// TwinCAT 3 PLC project TS_PLC
// ProgramVersion: 3.1.4024.0
// libraries:
//   Tc2_Standard, * (Beckhoff Automation GmbH)
//   Tc2_System, * (Beckhoff Automation GmbH)
//   Tc3_Module, * (Beckhoff Automation GmbH)
// project tree:
//   GVLs/ GVL_IO.TcGVL
//   / PlcTask.TcTTO, SimTask.TcTTO
//   POUs/FBs/ FB_Conveyor.TcPOU, FB_Init.TcPOU, FB_LTU.TcPOU, FB_MotorUnit.TcPOU, FB_Reader.TcPOU, FB_Stopper.TcPOU
//   POUs/FBs/Homing/ FB_HomingLTU.TcPOU, FB_HomingManager.TcPOU
//   POUs/FBs/Interchange/ FB_TransferChain_LowerToUpper.TcPOU, FB_TransferChain_UpperToLower.TcPOU, FB_TransferCorner_LowerToUpper.TcPOU, FB_TransferCorner_UpperToLower.TcPOU, FB_DirectTransferGreen.TcPOU, FB_DirectTransferOrange.TcPOU
//   POUs/FBs/Scheduler/ FB_Scheduler.TcPOU, FB_Scheduler_Queue.TcPOU, FB_Scheduler_Queue_copy.TcPOU, FB_ThroughputMonitor.TcPOU
//   POUs/FCs/ FB_AutoPlace.TcPOU
//   POUs/ MAIN.TcPOU, PRG_SIM.TcPOU
//   POUs/Simulation/ FB_InjectAfterRelease.TcPOU, FB_SimConveyor.TcPOU, FB_SimLTU.TcPOU, FB_SimReader.TcPOU, FB_SimStopper.TcPOU
// real-time tasks:
//   TASK PlcTask: cycle T#10ms, priority 20, ADS port 350
//   TASK SimTask: cycle T#10ms, priority 1, ADS port 351
// variable links:
//   TS_PLC/TS_PLC Instance <-> TS_PLC/TS_PLC Instance
//     PlcTask Inputs/MAIN.Conv12_6.MotorOK <-> SimTask Outputs/PRG_SIM.SimConv12_6.MotorOK
//     PlcTask Inputs/MAIN.Conv3_9.MotorOK <-> SimTask Outputs/PRG_SIM.SimConv3_9.MotorOK
//     PlcTask Inputs/MAIN.Conv6_12.MotorOK <-> SimTask Outputs/PRG_SIM.SimConv6_12.MotorOK
//     PlcTask Inputs/MAIN.Conv9_3.MotorOK <-> SimTask Outputs/PRG_SIM.SimConv9_3.MotorOK
//     PlcTask Inputs/MAIN.Conv12_6.RunningIn <-> SimTask Outputs/PRG_SIM.SimConv12_6.RunningIn
//     PlcTask Inputs/MAIN.Conv3_9.RunningIn <-> SimTask Outputs/PRG_SIM.SimConv3_9.RunningIn
//     PlcTask Inputs/MAIN.Conv6_12.RunningIn <-> SimTask Outputs/PRG_SIM.SimConv6_12.RunningIn
//     PlcTask Inputs/MAIN.Conv9_3.RunningIn <-> SimTask Outputs/PRG_SIM.SimConv9_3.RunningIn
//     PlcTask Inputs/MAIN.LTU_12_3.MotorOK <-> SimTask Outputs/PRG_SIM.SimLTU12_3.MotorOK
//     PlcTask Inputs/MAIN.LTU_3_6.MotorOK <-> SimTask Outputs/PRG_SIM.SimLTU3_6.MotorOK
//     PlcTask Inputs/MAIN.LTU_6_9.MotorOK <-> SimTask Outputs/PRG_SIM.SimLTU6_9.MotorOK
//     PlcTask Inputs/MAIN.LTU_9_12.MotorOK <-> SimTask Outputs/PRG_SIM.SimLTU9_12.MotorOK
//     PlcTask Inputs/MAIN.LTU_12_3.PosBottomIn <-> SimTask Outputs/PRG_SIM.SimLTU12_3.PosBottom
//     PlcTask Inputs/MAIN.LTU_3_6.PosBottomIn <-> SimTask Outputs/PRG_SIM.SimLTU3_6.PosBottom
//     PlcTask Inputs/MAIN.LTU_6_9.PosBottomIn <-> SimTask Outputs/PRG_SIM.SimLTU6_9.PosBottom
//     PlcTask Inputs/MAIN.LTU_9_12.PosBottomIn <-> SimTask Outputs/PRG_SIM.SimLTU9_12.PosBottom
//     PlcTask Inputs/MAIN.LTU_12_3.PosMidIn <-> SimTask Outputs/PRG_SIM.SimLTU12_3.PosMid
//     PlcTask Inputs/MAIN.LTU_3_6.PosMidIn <-> SimTask Outputs/PRG_SIM.SimLTU3_6.PosMid
//     PlcTask Inputs/MAIN.LTU_6_9.PosMidIn <-> SimTask Outputs/PRG_SIM.SimLTU6_9.PosMid
//     PlcTask Inputs/MAIN.LTU_9_12.PosMidIn <-> SimTask Outputs/PRG_SIM.SimLTU9_12.PosMid
//     PlcTask Inputs/MAIN.LTU_12_3.PosTopIn <-> SimTask Outputs/PRG_SIM.SimLTU12_3.PosTop
//     PlcTask Inputs/MAIN.LTU_3_6.PosTopIn <-> SimTask Outputs/PRG_SIM.SimLTU3_6.PosTop
//     PlcTask Inputs/MAIN.LTU_6_9.PosTopIn <-> SimTask Outputs/PRG_SIM.SimLTU6_9.PosTop
//     PlcTask Inputs/MAIN.LTU_9_12.PosTopIn <-> SimTask Outputs/PRG_SIM.SimLTU9_12.PosTop
//     PlcTask Inputs/MAIN.LTU_12_3.RunningIn <-> SimTask Outputs/PRG_SIM.SimLTU12_3.PushRunning
//     PlcTask Inputs/MAIN.LTU_3_6.RunningIn <-> SimTask Outputs/PRG_SIM.SimLTU3_6.PushRunning
//     PlcTask Inputs/MAIN.LTU_6_9.RunningIn <-> SimTask Outputs/PRG_SIM.SimLTU6_9.PushRunning
//     PlcTask Inputs/MAIN.LTU_9_12.RunningIn <-> SimTask Outputs/PRG_SIM.SimLTU9_12.PushRunning
//     PlcTask Inputs/MAIN.Reader{3..12 step 3}.I_ReaderValue <-> SimTask Outputs/PRG_SIM.SimReader_{3..12 step 3}.ReaderValue  (4 links)
//     SimTask Inputs/PRG_SIM.SimBlue{3..12 step 3}.CarrierIn <-> PlcTask Outputs/MAIN.Reader{3..12 step 3}.Valid  (4 links)
//     SimTask Inputs/PRG_SIM.SimBlue{3..12 step 3}.CmdDown <-> PlcTask Outputs/MAIN.Blue{3..12 step 3}.StopperDown  (4 links)
//     SimTask Inputs/PRG_SIM.SimConv12_6.MotorRun <-> PlcTask Outputs/MAIN.Conv12_6.MotorRun
//     SimTask Inputs/PRG_SIM.SimConv3_9.MotorRun <-> PlcTask Outputs/MAIN.Conv3_9.MotorRun
//     SimTask Inputs/PRG_SIM.SimConv6_12.MotorRun <-> PlcTask Outputs/MAIN.Conv6_12.MotorRun
//     SimTask Inputs/PRG_SIM.SimConv9_3.MotorRun <-> PlcTask Outputs/MAIN.Conv9_3.MotorRun
//     SimTask Inputs/PRG_SIM.SimLTU12_3.CmdPush <-> PlcTask Outputs/MAIN.LTU_12_3.LTU_MotorRun
//     SimTask Inputs/PRG_SIM.SimLTU3_6.CmdPush <-> PlcTask Outputs/MAIN.LTU_3_6.LTU_MotorRun
//     SimTask Inputs/PRG_SIM.SimLTU6_9.CmdPush <-> PlcTask Outputs/MAIN.LTU_6_9.LTU_MotorRun
//     SimTask Inputs/PRG_SIM.SimLTU9_12.CmdPush <-> PlcTask Outputs/MAIN.LTU_9_12.LTU_MotorRun
//     SimTask Inputs/PRG_SIM.SimLTU12_3.MoveDown <-> PlcTask Outputs/MAIN.LTU_12_3.CylToBottom
//     SimTask Inputs/PRG_SIM.SimLTU3_6.MoveDown <-> PlcTask Outputs/MAIN.LTU_3_6.CylToBottom
//     SimTask Inputs/PRG_SIM.SimLTU6_9.MoveDown <-> PlcTask Outputs/MAIN.LTU_6_9.CylToBottom
//     SimTask Inputs/PRG_SIM.SimLTU9_12.MoveDown <-> PlcTask Outputs/MAIN.LTU_9_12.CylToBottom
//     SimTask Inputs/PRG_SIM.SimLTU12_3.MoveUp <-> PlcTask Outputs/MAIN.LTU_12_3.CylToTop
//     SimTask Inputs/PRG_SIM.SimLTU3_6.MoveUp <-> PlcTask Outputs/MAIN.LTU_3_6.CylToTop
//     SimTask Inputs/PRG_SIM.SimLTU6_9.MoveUp <-> PlcTask Outputs/MAIN.LTU_6_9.CylToTop
//     SimTask Inputs/PRG_SIM.SimLTU9_12.MoveUp <-> PlcTask Outputs/MAIN.LTU_9_12.CylToTop
//     SimTask Inputs/PRG_SIM.SimPurp3_9_1.CmdDown <-> PlcTask Outputs/MAIN.Purple3_9_1.StopperDown
//     SimTask Inputs/PRG_SIM.SimPurp3_9_2.CmdDown <-> PlcTask Outputs/MAIN.Purple3_9_2.StopperDown
//     SimTask Inputs/PRG_SIM.SimPurp9_3_1.CmdDown <-> PlcTask Outputs/MAIN.Purple9_3_1.StopperDown
//     SimTask Inputs/PRG_SIM.SimPurp9_3_2.CmdDown <-> PlcTask Outputs/MAIN.Purple9_3_2.StopperDown
//     SimTask Inputs/PRG_SIM.SimReader_{3..12 step 3}.TriggerRead <-> PlcTask Outputs/MAIN.Reader{3..12 step 3}.vTrigger  (4 links)

CONFIGURATION TS_PLC
    RESOURCE PLC ON TwinCAT3
        TASK PlcTask(INTERVAL := T#10ms, PRIORITY := 20);
        TASK SimTask(INTERVAL := T#10ms, PRIORITY := 1);
        PROGRAM MAIN WITH PlcTask : MAIN;
        PROGRAM PRG_SIM WITH SimTask : PRG_SIM;
    END_RESOURCE
END_CONFIGURATION

// ---- GVLs/GVL_IO.TcGVL
{attribute 'qualified_only'}
VAR_GLOBAL
	//
END_VAR

// ---- POUs/MAIN.TcPOU
PROGRAM MAIN
VAR
	InitFB : FB_Init;
	
	Conv12_6 : FB_Conveyor;
	Conv6_12 : FB_Conveyor;
	Conv3_9 : FB_Conveyor;
	Conv9_3 : FB_Conveyor;
	
	Blue12 : FB_Stopper;
	Blue6 : FB_Stopper;
	Blue3 : FB_Stopper;
	Blue9 : FB_Stopper;
	
	LTU_12_3 : FB_LTU;
	LTU_3_6 : FB_LTU;
	LTU_6_9 : FB_LTU;
	LTU_9_12 : FB_LTU;
	
	Purple9_3_1 : FB_Stopper;
	Purple9_3_2 : FB_Stopper;
	Purple3_9_1 : FB_Stopper;
	Purple3_9_2 : FB_Stopper;
	
	Reader12 : FB_Reader;
	Reader3 : FB_Reader;
	Reader6 : FB_Reader;
	Reader9 : FB_Reader;
	tPulse : TP;
	tPulse1 : TP;
	startRead: BOOL;
	
	
	Blue12_Occupied: BOOL;
	LTU_3_6_LightBarrierIn: BOOL;
	LTU_12_3_LightBarrierIn: BOOL;
	
	Blue6_Occupied: BOOL;
	LTU_6_9_LightBarrierIn: BOOL;
	LTU_9_12_LightBarrierIn: BOOL;
	
	
	Blue9_Occupied: BOOL;
	Purple9_3_1_Occ: BOOL;
	Purple9_3_2_Occ: BOOL;
	
	//Scheduler : FB_Scheduler;
	Scheduler : FB_Scheduler_Queue;
	
	Transfer_12_6 : FB_DirectTransferGreen;
	Transfer_6_12 : FB_DirectTransferGreen;
	
	Transfer_9_3 : FB_DirectTransferOrange;
	Transfer_3_9 : FB_DirectTransferOrange;
	
	Transfer_12_3 : FB_TransferCorner_LowerToUpper;
	Transfer_6_9 : FB_TransferCorner_LowerToUpper;
	Transfer_3_6 : FB_TransferCorner_UpperToLower;
	Transfer_9_12 : FB_TransferCorner_UpperToLower;
	
	Transfer_12_9 : FB_TransferChain_LowerToUpper;
	Transfer_6_3 : FB_TransferChain_LowerToUpper;
	Transfer_9_6 : FB_TransferChain_UpperToLower;
	Transfer_3_12 : FB_TransferChain_UpperToLower;
	
	Throughput : FB_ThroughputMonitor;
	HomingMgr : FB_HomingManager;
	
	DebugWhoWroteBlue6: STRING(128);
	AllLTUsHomed: BOOL;
	HomingError: BOOL;
	ResetGlobal: BOOL;
	SchedulerBusy: BOOL;
	SchedulerQCount: INT;
	StartHomingGlobal: BOOL;
	OnTimer : ton;
	Start: BOOL;
	Auto_Reader12 : FB_AutoPlace;
END_VAR

InitFB(
    Reset     := ,   // manual reset button/flag
    Blue12    := Blue12,
    Blue3     := Blue3,
    Blue6     := Blue6,
    Blue9     := Blue9,
    Purple9_3_1 := Purple9_3_1,
    Purple9_3_2 := Purple9_3_2,
    Purple3_9_1 := Purple3_9_1,
    Purple3_9_2 := Purple3_9_2,
    LTU_12_3 := LTU_12_3,
    LTU_3_6  := LTU_3_6,
    LTU_6_9  := LTU_6_9,
    LTU_9_12 := LTU_9_12,
    Scheduler := Scheduler
);
IF AllLTUsHomed THEN
	Auto_Reader12(BlueStopper:= Blue12.CmdDown, Reader_Trigger=> Reader12.TriggerRead);
END_IF
Conv12_6(
	CmdRunRequest:= TRUE, 
	MotorOK:= , 
	RunningIn:= , 
	PathClear:= TRUE, 
	MotorRun=> , 
	IsRunning=> );
	
Conv6_12(
	CmdRunRequest:= TRUE, 
	MotorOK:= , 
	RunningIn:= , 
	PathClear:= TRUE, 
	MotorRun=> , 
	IsRunning=> );

Conv3_9(
	CmdRunRequest:= TRUE, 
	MotorOK:= , 
	RunningIn:= , 
	PathClear:= TRUE, 
	MotorRun=> , 
	IsRunning=> );
	
Conv9_3(
	CmdRunRequest:= TRUE, 
	MotorOK:= , 
	RunningIn:= , 
	PathClear:= TRUE, 
	MotorRun=> , 
	IsRunning=> );


	
Blue12(CmdDown:= , OccupiedIn:= , StopperDown=> , Occupied=> );
Blue6(CmdDown:= , OccupiedIn:= , StopperDown=> , Occupied=> );
Blue3(CmdDown:= , OccupiedIn:= , StopperDown=> , Occupied=> );
Blue9(CmdDown:= , OccupiedIn:= , StopperDown=> , Occupied=> );

LTU_12_3(
	CmdMoveUp:= , 
	CmdMoveDown:= ,  
	MotorOK:= , 
	RunningIn:= , 
	LightBarrierIn:= , 
	PosBottomIn:= , 
	PosMidIn:= , 
	PosTopIn:= , 
	CylToTop=> , 
	CylToBottom=> , 
	LTU_MotorRun=> , 
	IsRunning=> , 
	PosBottom=> , 
	PosMid=> , 
	PosTop=> , 
	IsFree=> );
	
LTU_3_6(
	CmdMoveUp:= , 
	CmdMoveDown:= ,  
	MotorOK:= , 
	RunningIn:= , 
	LightBarrierIn:= , 
	PosBottomIn:= , 
	PosMidIn:= , 
	PosTopIn:= , 
	CylToTop=> , 
	CylToBottom=> , 
	LTU_MotorRun=> , 
	IsRunning=> , 
	PosBottom=> , 
	PosMid=> , 
	PosTop=> , 
	IsFree=> );
LTU_6_9(
	CmdMoveUp:= , 
	CmdMoveDown:= ,  
	MotorOK:= , 
	RunningIn:= , 
	LightBarrierIn:= , 
	PosBottomIn:= , 
	PosMidIn:= , 
	PosTopIn:= , 
	CylToTop=> , 
	CylToBottom=> , 
	LTU_MotorRun=> , 
	IsRunning=> , 
	PosBottom=> , 
	PosMid=> , 
	PosTop=> , 
	IsFree=> );
LTU_9_12(
	CmdMoveUp:= , 
	CmdMoveDown:= ,  
	MotorOK:= , 
	RunningIn:= , 
	LightBarrierIn:= , 
	PosBottomIn:= , 
	PosMidIn:= , 
	PosTopIn:= , 
	CylToTop=> , 
	CylToBottom=> , 
	LTU_MotorRun=> , 
	IsRunning=> , 
	PosBottom=> , 
	PosMid=> , 
	PosTop=> , 
	IsFree=> );
	
Purple9_3_1(CmdDown:= , OccupiedIn:= , StopperDown=> , Occupied=> );
Purple9_3_2(CmdDown:= , OccupiedIn:= , StopperDown=> , Occupied=> );
Purple3_9_1(CmdDown:= , OccupiedIn:= , StopperDown=> , Occupied=> );
Purple3_9_2(CmdDown:= , OccupiedIn:= , StopperDown=> , Occupied=> );	

	
Reader12(TriggerRead:= ,Dest:=6,Source:=12, ReaderValue=> , Valid=> );	
Reader3(TriggerRead:= ,Dest:=6,Source:=3, ReaderValue=> , Valid=> );	
Reader6(TriggerRead:= ,Dest:=9,Source:=6, ReaderValue=> , Valid=> );	
Reader9(TriggerRead:= ,Dest:=6,Source:=9, ReaderValue=> , Valid=> );	

// === Homing Manager ===
HomingMgr(
    StartHoming := StartHomingGlobal,   // your button / auto-start flag
    Reset       := ,         // global reset button

    LTU_12_3_PosTop    := LTU_12_3.PosTop,
    LTU_12_3_PosBottom := LTU_12_3.PosBottom,
    LTU_12_3_PosMid    := LTU_12_3.PosMid,
    LTU_12_3_Running   := LTU_12_3.IsRunning,

    LTU_3_6_PosTop    := LTU_3_6.PosTop,
    LTU_3_6_PosBottom := LTU_3_6.PosBottom,
    LTU_3_6_PosMid    := LTU_3_6.PosMid,
    LTU_3_6_Running   := LTU_3_6.IsRunning,

    LTU_9_12_PosTop    := LTU_9_12.PosTop,
    LTU_9_12_PosBottom := LTU_9_12.PosBottom,
    LTU_9_12_PosMid    := LTU_9_12.PosMid,
    LTU_9_12_Running   := LTU_9_12.IsRunning,

    LTU_6_9_PosTop    := LTU_6_9.PosTop,
    LTU_6_9_PosBottom := LTU_6_9.PosBottom,
    LTU_6_9_PosMid    := LTU_6_9.PosMid,
    LTU_6_9_Running   := LTU_6_9.IsRunning,

    LTU_12_3_CmdMoveUp   => LTU_12_3.CmdMoveUp,
    LTU_12_3_CmdMoveDown => LTU_12_3.CmdMoveDown,

    LTU_3_6_CmdMoveUp   => LTU_3_6.CmdMoveUp,
    LTU_3_6_CmdMoveDown => LTU_3_6.CmdMoveDown,

    LTU_9_12_CmdMoveUp   => LTU_9_12.CmdMoveUp,
    LTU_9_12_CmdMoveDown => LTU_9_12.CmdMoveDown,

    LTU_6_9_CmdMoveUp   => LTU_6_9.CmdMoveUp,
    LTU_6_9_CmdMoveDown => LTU_6_9.CmdMoveDown,

    AllDone   => AllLTUsHomed,
    AnyError  => HomingError
);

// === Scheduler (enabled only after homing) ===
IF AllLTUsHomed AND NOT HomingError THEN
    Scheduler(
        Reader12_Valid := Reader12.Valid,
        Reader12_Value := Reader12.ReaderValue,
        Reader3_Valid  := Reader3.Valid,
        Reader3_Value  := Reader3.ReaderValue,
        Reader6_Valid  := Reader6.Valid,
        Reader6_Value  := Reader6.ReaderValue,
        Reader9_Valid  := Reader9.Valid,
        Reader9_Value  := Reader9.ReaderValue,

        // Done flags from all transfers
        T12_6_Done := Transfer_12_6.Done,
        T6_12_Done := Transfer_6_12.Done,
        T9_3_Done  := Transfer_9_3.Done,
        T3_9_Done  := Transfer_3_9.Done,
        T12_3_Done := Transfer_12_3.Done,
        T6_9_Done  := Transfer_6_9.Done,
        T3_6_Done  := Transfer_3_6.Done,
        T9_12_Done := Transfer_9_12.Done,
        T12_9_Done := Transfer_12_9.Done,
        T6_3_Done  := Transfer_6_3.Done,
        T9_6_Done  := Transfer_9_6.Done,
        T3_12_Done := Transfer_3_12.Done,

        Reset := 
    );
ELSE
    // Prevent scheduler outputs until homed
    SchedulerBusy := FALSE;
END_IF


// Scheduler -- Only start a transfer if the system is free (no other active transfer)
// Run Scheduler
//Scheduler(
//    Reader12_Valid := Reader12.Valid,
//    Reader12_Value := Reader12.ReaderValue,
//    Reader3_Valid  := Reader3.Valid,
//    Reader3_Value  := Reader3.ReaderValue,
//    Reader6_Valid  := Reader6.Valid,
//    Reader6_Value  := Reader6.ReaderValue,
//    Reader9_Valid  := Reader9.Valid,
//    Reader9_Value  := Reader9.ReaderValue,

//    // pass Done flags from all transfer FBs
//    T12_6_Done := Transfer_12_6.Done,
//    T6_12_Done := Transfer_6_12.Done,
//    T9_3_Done  := Transfer_9_3.Done,
//    T3_9_Done  := Transfer_3_9.Done,
//    T12_3_Done := Transfer_12_3.Done,
//    T6_9_Done  := Transfer_6_9.Done,
//    T3_6_Done  := Transfer_3_6.Done,
//    T9_12_Done := Transfer_9_12.Done,
//    T12_9_Done := Transfer_12_9.Done,
//    T6_3_Done  := Transfer_6_3.Done,
//    T9_6_Done  := Transfer_9_6.Done,
//    T3_12_Done := Transfer_3_12.Done,

//    Reset := 
//);



CASE Scheduler.activeRoute OF
	//..................*** Direct Transfer Green or Lower
	126:Transfer_12_6(JobID := Scheduler.JobID_12_6,
		StartRequest := Scheduler.Start_12_6,
		LTU1_PosOK   := LTU_12_3.PosBottom,
		LTU1_Running := LTU_12_3.IsRunning,
		LTU1_LB      := LTU_12_3_LightBarrierIn,
		LTU2_PosOK   := LTU_3_6.PosBottom,
		LTU2_Running := LTU_3_6.IsRunning,
		LTU2_LB      := LTU_3_6_LightBarrierIn,
		BlueOcc      := Blue12_Occupied,
	
		BlueCmdDown  => Blue12.CmdDown,
		Done         => ,
		Error        => ,
		LTU1_MoveDown=> LTU_12_3.CmdMoveDown,
		LTU2_MoveDown=>	LTU_3_6.CmdMoveDown,
	);
	612:Transfer_6_12(JobID := Scheduler.JobID_6_12,
		StartRequest := Scheduler.Start_6_12,
		LTU1_PosOK   := LTU_6_9.PosBottom,
		LTU1_Running := LTU_6_9.IsRunning,
		LTU1_LB      := LTU_6_9_LightBarrierIn,
		LTU2_PosOK   := LTU_9_12.PosBottom,
		LTU2_Running := LTU_9_12.IsRunning,
		LTU2_LB      := LTU_9_12_LightBarrierIn,
		BlueOcc      := Blue6_Occupied,
	
		BlueCmdDown  => Blue6.CmdDown,
		Done         => ,
		Error        => ,
		LTU1_MoveDown=> LTU_6_9.CmdMoveDown,
		LTU2_MoveDown=>	LTU_9_12.CmdMoveDown
	);
	DebugWhoWroteBlue6 := 'Transfer_6_12';
	//.................*** Direct Transfer Orange or Upper
	93:Transfer_9_3(JobID := Scheduler.JobID_9_3,
		StartRequest:= Scheduler.Start_9_3, 
		LTU1_PosOK:= LTU_9_12.PosTop, 
		LTU1_Running:= LTU_9_12.IsRunning, 
		LTU1_LB:= LTU_9_12_LightBarrierIn, 
		LTU2_PosOK:= LTU_12_3.PosTop, 
		LTU2_Running:= LTU_12_3.IsRunning, 
		LTU2_LB:= LTU_12_3_LightBarrierIn, 
		BlueOcc:= Blue9_Occupied, 
		Purple1Occ:= Purple9_3_1_Occ, 
		Purple2Occ:= Purple9_3_2_Occ, 
		reset:= , 
		BlueCmdDown=> Blue9.CmdDown, 
		Purple1CmdDown=> Purple9_3_1.CmdDown, 
		Purple2CmdDown=> Purple9_3_2.CmdDown, 
		LTU1_MoveUp=> LTU_9_12.CmdMoveUp, 
		LTU2_MoveUp=> LTU_12_3.CmdMoveUp, 
		Done=> , 
		Error=> 
	);
	
	39:Transfer_3_9(JobID := Scheduler.JobID_3_9,
		StartRequest := Scheduler.Start_3_9,
	
		// LTU_3_6
		LTU1_PosOK   := LTU_3_6.PosTop,
		LTU1_Running := LTU_3_6.IsRunning,
		LTU1_LB      := LTU_3_6.LightBarrierIn,
	
		// LTU_6_9
		LTU2_PosOK   := LTU_6_9.PosTop,
		LTU2_Running := LTU_6_9.IsRunning,
		LTU2_LB      := LTU_6_9.LightBarrierIn,
	
		// Stoppers
		BlueOcc      := Blue3.OccupiedIn,
		Purple1Occ   := Purple3_9_1.OccupiedIn,
		Purple2Occ   := Purple3_9_2.OccupiedIn,
	
		reset        := ,
	
		// Outputs
		BlueCmdDown   => Blue3.CmdDown,
		Purple1CmdDown=> Purple3_9_1.CmdDown,
		Purple2CmdDown=> Purple3_9_2.CmdDown,
		LTU1_MoveUp   => LTU_3_6.CmdMoveUp,
		LTU2_MoveUp   => LTU_6_9.CmdMoveUp,
	
		Done  => ,
		Error => 
	);
	
	//.........*************lower to upper corner****************
	123:Transfer_12_3(JobID := Scheduler.JobID_12_3,
		StartRequest:= Scheduler.Start_12_3, 
		LTU_PosTop:= LTU_12_3.PosTop, 
		LTU_PosBottom:= LTU_12_3.PosBottom, 
		LTU_Running:= LTU_12_3.IsRunning, 
		LTU_LB:= LTU_12_3.LightBarrierIn, 
		BlueOcc:= Blue12.OccupiedIn, 
		PurpleOcc:= Purple9_3_2.OccupiedIn, 
		reset:= , 
		BlueCmdDown=> Blue12.CmdDown, 
		PurpleCmdDown=> Purple9_3_2.CmdDown, 
		LTU_MoveUp=> LTU_12_3.CmdMoveUp, 
		LTU_MoveDown=> LTU_12_3.CmdMoveDown, 
		LTU_CmdPush=> LTU_12_3.CmdRun, 
		Done=> , 
		Error=> );
		
	69:Transfer_6_9(JobID := Scheduler.JobID_6_9,
		StartRequest := Scheduler.Start_6_9,
	
		// LTU_6_9
		LTU_PosTop    := LTU_6_9.PosTop,
		LTU_PosBottom := LTU_6_9.PosBottom,
		LTU_Running   := LTU_6_9.IsRunning,
		LTU_LB        := LTU_6_9.LightBarrierIn,
	
		// Stoppers
		BlueOcc       := Blue6.OccupiedIn,
		PurpleOcc     := Purple3_9_2.OccupiedIn,
	
		reset         := ,
	
		// Outputs
		BlueCmdDown   => Blue6.CmdDown,
		PurpleCmdDown => Purple3_9_2.CmdDown,
		LTU_MoveUp    => LTU_6_9.CmdMoveUp,
		LTU_MoveDown  => LTU_6_9.CmdMoveDown,
		LTU_CmdPush   => LTU_6_9.CmdRun,
	
		Done          => ,
		Error         => 
	);
	DebugWhoWroteBlue6 := 'Transfer_6_9';
	//...........**************Upper to Lower Corner.............................
	36:Transfer_3_6(JobID := Scheduler.JobID_3_6,
		StartRequest  := Scheduler.Start_3_6,
	
		LTU_PosTop    := LTU_3_6.PosTop,
		LTU_PosBottom := LTU_3_6.PosBottom,
		LTU_Running   := LTU_3_6.IsRunning,
		LTU_LB        := LTU_3_6.LightBarrierIn,
	
		BlueOcc       := Blue3.OccupiedIn,
		PurpleOcc     := Purple3_9_1.OccupiedIn,
	
		reset         := ,             // or leave blank if you handle reset elsewhere
	
		BlueCmdDown   => Blue3.CmdDown,
		PurpleCmdDown => Purple3_9_1.CmdDown,
		LTU_MoveUp    => LTU_3_6.CmdMoveUp,
		LTU_MoveDown  => LTU_3_6.CmdMoveDown,
		LTU_CmdPush   => LTU_3_6.CmdRun,
	
		Done          => ,
		Error         => 
	);
	912:Transfer_9_12(JobID := Scheduler.JobID_9_12,
		StartRequest  := Scheduler.Start_9_12,
	
		LTU_PosTop    := LTU_9_12.PosTop,
		LTU_PosBottom := LTU_9_12.PosBottom,
		LTU_Running   := LTU_9_12.IsRunning,
		LTU_LB        := LTU_9_12.LightBarrierIn,
	
		BlueOcc       := Blue9.OccupiedIn,
		PurpleOcc     := Purple9_3_1.OccupiedIn,
	
		reset         := ,   // or hook up your reset signal
	
		BlueCmdDown   => Blue9.CmdDown,
		PurpleCmdDown => Purple9_3_1.CmdDown,
		LTU_MoveUp    => LTU_9_12.CmdMoveUp,
		LTU_MoveDown  => LTU_9_12.CmdMoveDown,
		LTU_CmdPush   => LTU_9_12.CmdRun,
	
		Done          => ,
		Error         => 
	);
	
	
	// ............ Multi-hop transfer (12 -> 9) .............................
	//.......Lower to Upper Chain transfer....................................
	129:Transfer_12_9(JobID := Scheduler.JobID_12_9,
		StartRequest  := Scheduler.Start_12_9,
		reset         := ,
	
		// Blue12
		BlueOcc       := Blue12.OccupiedIn,
	
		// LTU_12_3
		LTU1_PosBottom:= LTU_12_3.PosBottom,
		LTU1_PosTop   := LTU_12_3.PosTop,
		LTU1_Running  := LTU_12_3.IsRunning,
		LTU1_LB       := LTU_12_3.LightBarrierIn,
	
		// LTU_3_6
		LTU2_PosBottom:= LTU_3_6.PosBottom,
		LTU2_PosTop   := LTU_3_6.PosTop,
		LTU2_Running  := LTU_3_6.IsRunning,
		LTU2_LB       := LTU_3_6.LightBarrierIn,
	
		// LTU_6_9
		LTU3_PosBottom:= LTU_6_9.PosBottom,
		LTU3_PosTop   := LTU_6_9.PosTop,
		LTU3_Running  := LTU_6_9.IsRunning,
		LTU3_LB       := LTU_6_9.LightBarrierIn,
	
		// Purples
		Purple1_Occ   := Purple9_3_2.OccupiedIn,   // first purple in chain
		Purple2_Occ   := Purple3_9_1.OccupiedIn,   // middle purple
		Purple3_Occ   := Purple3_9_2.OccupiedIn,   // final purple at exit
	
		// Outputs
		BlueCmdDown   => Blue12.CmdDown,
		Purple1CmdDown=> Purple9_3_2.CmdDown,
		Purple2CmdDown=> Purple3_9_1.CmdDown,
		Purple3CmdDown=> Purple3_9_2.CmdDown,
	
		LTU1_CmdPush  => LTU_12_3.CmdRun,
		LTU1_MoveUp   => LTU_12_3.CmdMoveUp,
		LTU1_MoveDown => LTU_12_3.CmdMoveDown,
	
		LTU2_CmdPush  => LTU_3_6.CmdRun,
		LTU2_MoveUp   => LTU_3_6.CmdMoveUp,
		LTU2_MoveDown => LTU_3_6.CmdMoveDown,
	
		LTU3_CmdPush  => LTU_6_9.CmdRun,
		LTU3_MoveUp   => LTU_6_9.CmdMoveUp,
		LTU3_MoveDown => LTU_6_9.CmdMoveDown,
	
		Done          => ,
		Error         => 
	);
	63:Transfer_6_3(JobID := Scheduler.JobID_6_3,
		StartRequest  := Scheduler.Start_6_3,
		reset         := ,
	
		// Blue6
		BlueOcc       := Blue6.OccupiedIn,
	
		// LTU_6_9
		LTU1_PosBottom:= LTU_6_9.PosBottom,
		LTU1_PosTop   := LTU_6_9.PosTop,
		LTU1_Running  := LTU_6_9.IsRunning,
		LTU1_LB       := LTU_6_9.LightBarrierIn,
	
		// LTU_9_12
		LTU2_PosBottom:= LTU_9_12.PosBottom,
		LTU2_PosTop   := LTU_9_12.PosTop,
		LTU2_Running  := LTU_9_12.IsRunning,
		LTU2_LB       := LTU_9_12.LightBarrierIn,
	
		// LTU_12_3
		LTU3_PosBottom:= LTU_12_3.PosBottom,
		LTU3_PosTop   := LTU_12_3.PosTop,
		LTU3_Running  := LTU_12_3.IsRunning,
		LTU3_LB       := LTU_12_3.LightBarrierIn,
	
		// Purples
		Purple1_Occ   := Purple3_9_2.OccupiedIn,
		Purple2_Occ   := Purple9_3_1.OccupiedIn,
		Purple3_Occ   := Purple9_3_2.OccupiedIn,
	
		// Outputs
		BlueCmdDown   => Blue6.CmdDown,
		Purple1CmdDown=> Purple3_9_2.CmdDown,
		Purple2CmdDown=> Purple9_3_1.CmdDown,
		Purple3CmdDown=> Purple9_3_2.CmdDown,
	
		LTU1_CmdPush  => LTU_6_9.CmdRun,
		LTU1_MoveUp   => LTU_6_9.CmdMoveUp,
		LTU1_MoveDown => LTU_6_9.CmdMoveDown,
	
		LTU2_CmdPush  => LTU_9_12.CmdRun,
		LTU2_MoveUp   => LTU_9_12.CmdMoveUp,
		LTU2_MoveDown => LTU_9_12.CmdMoveDown,
	
		LTU3_CmdPush  => LTU_12_3.CmdRun,
		LTU3_MoveUp   => LTU_12_3.CmdMoveUp,
		LTU3_MoveDown => LTU_12_3.CmdMoveDown,
	
		Done          => ,
		Error         => 
	);
	DebugWhoWroteBlue6 := 'Transfer_6_3';
	
	//.......Upper to Lower Chain transfer....................................
	96:Transfer_9_6(JobID := Scheduler.JobID_9_6,
		StartRequest  := Scheduler.Start_9_6,
		reset         := ,
	
		// Blue9
		BlueOcc       := Blue9.OccupiedIn,
	
		// LTU_9_12
		LTU1_PosBottom:= LTU_9_12.PosBottom,
		LTU1_PosTop   := LTU_9_12.PosTop,
		LTU1_Running  := LTU_9_12.IsRunning,
		LTU1_LB       := LTU_9_12.LightBarrierIn,
	
		// LTU_12_3
		LTU2_PosBottom:= LTU_12_3.PosBottom,
		LTU2_PosTop   := LTU_12_3.PosTop,
		LTU2_Running  := LTU_12_3.IsRunning,
		LTU2_LB       := LTU_12_3.LightBarrierIn,
	
		// LTU_3_6
		LTU3_PosBottom:= LTU_3_6.PosBottom,
		LTU3_PosTop   := LTU_3_6.PosTop,
		LTU3_Running  := LTU_3_6.IsRunning,
		LTU3_LB       := LTU_3_6.LightBarrierIn,
	
		// Purples
		Purple1_Occ   := Purple9_3_1.OccupiedIn,   // first purple in path
		Purple2_Occ   := Purple9_3_2.OccupiedIn,   // second purple
	
		// Outputs
		BlueCmdDown   => Blue9.CmdDown,
		Purple1CmdDown=> Purple9_3_1.CmdDown,
		Purple2CmdDown=> Purple9_3_2.CmdDown,
	
		LTU1_CmdPush  => LTU_9_12.CmdRun,
		LTU1_MoveUp   => LTU_9_12.CmdMoveUp,
		LTU1_MoveDown => LTU_9_12.CmdMoveDown,
	
		LTU2_CmdPush  => LTU_12_3.CmdRun,
		LTU2_MoveUp   => LTU_12_3.CmdMoveUp,
		LTU2_MoveDown => LTU_12_3.CmdMoveDown,
	
		LTU3_CmdPush  => LTU_3_6.CmdRun,
		LTU3_MoveUp   => LTU_3_6.CmdMoveUp,
		LTU3_MoveDown => LTU_3_6.CmdMoveDown,
	
		Done          => ,
		Error         => 
	);	
	312:Transfer_3_12(JobID := Scheduler.JobID_3_12,
		StartRequest  := Scheduler.Start_3_12,
		reset         := ,
	
		// Blue3
		BlueOcc       := Blue3.OccupiedIn,
	
		// LTU_3_6
		LTU1_PosBottom:= LTU_3_6.PosBottom,
		LTU1_PosTop   := LTU_3_6.PosTop,
		LTU1_Running  := LTU_3_6.IsRunning,
		LTU1_LB       := LTU_3_6.LightBarrierIn,
	
		// LTU_6_9
		LTU2_PosBottom:= LTU_6_9.PosBottom,
		LTU2_PosTop   := LTU_6_9.PosTop,
		LTU2_Running  := LTU_6_9.IsRunning,
		LTU2_LB       := LTU_6_9.LightBarrierIn,
	
		// LTU_9_12
		LTU3_PosBottom:= LTU_9_12.PosBottom,
		LTU3_PosTop   := LTU_9_12.PosTop,
		LTU3_Running  := LTU_9_12.IsRunning,
		LTU3_LB       := LTU_9_12.LightBarrierIn,
	
		// Purples
		Purple1_Occ   := Purple3_9_1.OccupiedIn,
		Purple2_Occ   := Purple3_9_2.OccupiedIn,
		Purple3_Occ   := Purple9_3_1.OccupiedIn,
	
		// Outputs
		BlueCmdDown   => Blue3.CmdDown,
		Purple1CmdDown=> Purple3_9_1.CmdDown,
		Purple2CmdDown=> Purple3_9_2.CmdDown,
		Purple3CmdDown=> Purple9_3_1.CmdDown,
	
		LTU1_CmdPush  => LTU_3_6.CmdRun,
		LTU1_MoveUp   => LTU_3_6.CmdMoveUp,
		LTU1_MoveDown => LTU_3_6.CmdMoveDown,
	
		LTU2_CmdPush  => LTU_6_9.CmdRun,
		LTU2_MoveUp   => LTU_6_9.CmdMoveUp,
		LTU2_MoveDown => LTU_6_9.CmdMoveDown,
	
		LTU3_CmdPush  => LTU_9_12.CmdRun,
		LTU3_MoveUp   => LTU_9_12.CmdMoveUp,
		LTU3_MoveDown => LTU_9_12.CmdMoveDown,
	
		Done          => ,
		Error         => 
	);
ELSE
    // no active route → don’t call any transfer FB
	//DebugWhoWroteBlue6 := 'NONE';
END_CASE


Throughput(
    DonePulse := (
        Transfer_12_6.Done OR
        Transfer_6_12.Done OR
        Transfer_9_3.Done  OR
        Transfer_3_9.Done  OR
        Transfer_12_3.Done OR
        Transfer_6_9.Done  OR
        Transfer_3_6.Done  OR
        Transfer_9_12.Done OR
        Transfer_12_9.Done OR
        Transfer_6_3.Done  OR
        Transfer_9_6.Done  OR
        Transfer_3_12.Done
    ),
    Reset := 
);

END_PROGRAM

// ---- POUs/FBs/FB_Init.TcPOU
FUNCTION_BLOCK FB_Init
VAR_INPUT
    Reset : BOOL;   // external reset (button/flag)
END_VAR
VAR_IN_OUT
    Blue12, Blue3, Blue6, Blue9 : FB_Stopper;
    Purple9_3_1, Purple9_3_2, Purple3_9_1, Purple3_9_2 : FB_Stopper;
    LTU_12_3, LTU_3_6, LTU_6_9, LTU_9_12 : FB_LTU;
    Scheduler : FB_Scheduler_Queue;
END_VAR
VAR
    firstScan : BOOL := TRUE;   // internal latch
END_VAR

// --- Safe State Logic ---
IF firstScan OR Reset THEN
    // Blue stoppers (all blocking)
    Blue12.CmdDown := TRUE;
    Blue3.CmdDown  := TRUE;
    Blue6.CmdDown  := TRUE;
    Blue9.CmdDown  := TRUE;

    // Purple stoppers (all blocking)
    Purple9_3_1.CmdDown := TRUE;
    Purple9_3_2.CmdDown := TRUE;
    Purple3_9_1.CmdDown := TRUE;
    Purple3_9_2.CmdDown := TRUE;

    // LTUs (all idle)
    LTU_12_3.CmdMoveUp   := FALSE;
    LTU_12_3.CmdMoveDown := FALSE;
    LTU_12_3.CmdRun      := FALSE;

    LTU_3_6.CmdMoveUp    := FALSE;
    LTU_3_6.CmdMoveDown  := FALSE;
    LTU_3_6.CmdRun       := FALSE;

    LTU_6_9.CmdMoveUp    := FALSE;
    LTU_6_9.CmdMoveDown  := FALSE;
    LTU_6_9.CmdRun       := FALSE;

    LTU_9_12.CmdMoveUp   := FALSE;
    LTU_9_12.CmdMoveDown := FALSE;
    LTU_9_12.CmdRun      := FALSE;

    // Tell Scheduler to reset itself
    Scheduler(Reset := TRUE);

    // clear firstScan latch
    firstScan := FALSE;
ELSE
    // normal scheduler call, Reset=FALSE
    Scheduler(Reset := FALSE);
END_IF

END_FUNCTION_BLOCK

// ---- POUs/FBs/FB_Stopper.TcPOU
FUNCTION_BLOCK FB_Stopper
VAR_INPUT
    CmdDown   : BOOL;   // TRUE = stopper down (block carrier)
    OccupiedIn AT%I*: BOOL;   // Sensor input
END_VAR
VAR_OUTPUT
    StopperDown AT%Q*: BOOL; // Actuator output
    Occupied    : BOOL; // Output copy of sensor
END_VAR

// Direct assignments
StopperDown := CmdDown;
Occupied    := OccupiedIn;

END_FUNCTION_BLOCK

// ---- POUs/FBs/FB_LTU.TcPOU
FUNCTION_BLOCK FB_LTU
VAR_INPUT
    CmdMoveUp      : BOOL;   // request cylinder to Top
    CmdMoveDown    : BOOL;   // request cylinder to Bottom
    CmdRun         : BOOL;   // run LTU motor
    MotorOK        AT%I*: BOOL;
    RunningIn      AT%I*: BOOL;   // motor running feedback
    LightBarrierIn AT%I*: BOOL;   // TRUE if LTU free
    PosBottomIn    AT%I*: BOOL;
    PosMidIn       AT%I*: BOOL;
    PosTopIn       AT%I*: BOOL;
END_VAR
VAR_OUTPUT
    CylToTop       AT%Q*: BOOL;   // actuator output
    CylToBottom    AT%Q*: BOOL;   // actuator output
    LTU_MotorRun   AT%Q*: BOOL;   // actuator output
    IsRunning      : BOOL;   // motor running feedback
    PosBottom      : BOOL;
    PosMid         : BOOL;
    PosTop         : BOOL;
    IsFree         : BOOL;   // derived from LightBarrierIn
END_VAR
VAR
    Motor : FB_MotorUnit;
END_VAR

// Cylinder logic (safe mutual exclusion)
CylToTop    := CmdMoveUp AND NOT CmdMoveDown;
CylToBottom := CmdMoveDown AND NOT CmdMoveUp;

// Motor logic
Motor(CmdRun := CmdRun,
      MotorOK := MotorOK,
      RunningIn := RunningIn);

LTU_MotorRun := Motor.MotorRun;
IsRunning    := Motor.IsRunning;

// Pass-through sensors
PosBottom := PosBottomIn;
PosMid    := PosMidIn;
PosTop    := PosTopIn;
IsFree    := LightBarrierIn;

END_FUNCTION_BLOCK

// ---- POUs/FBs/FB_MotorUnit.TcPOU
FUNCTION_BLOCK FB_MotorUnit
VAR_INPUT
    CmdRun   : BOOL;   // Command from controller
    MotorOK  : BOOL;   // from sensor Motor health input
	RunningIn : BOOL;  // From sensor (conveyor running feedback)
END_VAR
VAR_OUTPUT
    MotorRun : BOOL;   // Output to motor actuator
    IsRunning: BOOL;   // Sensor input: motor running
END_VAR
VAR
    //
END_VAR

// Simple interlock
MotorRun   := CmdRun AND MotorOK ;
IsRunning  := RunningIn;

END_FUNCTION_BLOCK

// ---- POUs/FBs/Scheduler/FB_Scheduler_Queue.TcPOU
FUNCTION_BLOCK FB_Scheduler_Queue
VAR_INPUT
    // Reader inputs
    Reader12_Valid : BOOL;
    Reader12_Value : INT;
    Reader3_Valid  : BOOL;
    Reader3_Value  : INT;
    Reader6_Valid  : BOOL;
    Reader6_Value  : INT;
    Reader9_Valid  : BOOL;
    Reader9_Value  : INT;

    // Done flags from transfers
    T12_6_Done, T6_12_Done : BOOL;
    T9_3_Done,  T3_9_Done  : BOOL;
    T12_3_Done, T6_9_Done  : BOOL;
    T3_6_Done,  T9_12_Done : BOOL;
    T12_9_Done, T6_3_Done  : BOOL;
    T9_6_Done,  T3_12_Done : BOOL;

    Reset : BOOL;
END_VAR
VAR_OUTPUT
    // Start signals (1-scan pulses)
    Start_12_6, Start_6_12 : BOOL;
    Start_9_3,  Start_3_9  : BOOL;
    Start_12_3, Start_6_9  : BOOL;
    Start_3_6,  Start_9_12 : BOOL;
    Start_12_9, Start_6_3  : BOOL;
    Start_9_6,  Start_3_12 : BOOL;

    Busy        : BOOL;
    QCount      : INT;     // number of queued requests
    activeRoute : INT;     // currently executing route
END_VAR
VAR
    queue   : ARRAY[1..10] OF INT;   // FIFO buffer (10 deep)
    head    : INT := 1;
    tail    : INT := 1;
	prevR12, prevR3, prevR6, prevR9 : BOOL;
END_VAR

// === Reset ===
IF Reset THEN
    head := 1; tail := 1; QCount := 0;
    Busy := FALSE; activeRoute := 0;
END_IF

// === Enqueue new reader requests ===
IF Reader12_Valid AND NOT prevR12 THEN
    CASE Reader12_Value OF
        6: Enqueue(126);
        3: Enqueue(123);
        9: Enqueue(129);
    END_CASE
END_IF
prevR12 := Reader12_Valid;

IF Reader6_Valid AND NOT prevR6 THEN
    CASE Reader6_Value OF
        12: Enqueue(612);
        9:  Enqueue(69);
        3:  Enqueue(63);
    END_CASE
END_IF
prevR6 := Reader6_Valid;

IF Reader3_Valid AND NOT prevR3 THEN
    CASE Reader3_Value OF
        9:  Enqueue(39);
        6:  Enqueue(36);
        12: Enqueue(312);
    END_CASE
END_IF
prevR3 := Reader3_Valid;

IF Reader9_Valid AND NOT prevR9 THEN
    CASE Reader9_Value OF
        3:  Enqueue(93);
        12: Enqueue(912);
        6:  Enqueue(96);
    END_CASE
END_IF
prevR9 := Reader9_Valid;


// === Dispatch logic ===
IF NOT Busy AND QCount > 0 THEN
    activeRoute := queue[head];
    head := (head MOD 10) + 1;
    QCount := QCount - 1;
    Busy := TRUE;

    // one-shot Start signal
    CASE activeRoute OF
        126: Start_12_6 := TRUE;
        612: Start_6_12 := TRUE;
        93 : Start_9_3  := TRUE;
        39 : Start_3_9  := TRUE;
        123: Start_12_3 := TRUE;
        69 : Start_6_9  := TRUE;
        36 : Start_3_6  := TRUE;
        912: Start_9_12 := TRUE;
        129: Start_12_9 := TRUE;
        63 : Start_6_3  := TRUE;
        96 : Start_9_6  := TRUE;
        312: Start_3_12 := TRUE;
    END_CASE
ELSE
    Start_12_6 := FALSE; Start_6_12 := FALSE;
    Start_9_3  := FALSE; Start_3_9  := FALSE;
    Start_12_3 := FALSE; Start_6_9  := FALSE;
    Start_3_6  := FALSE; Start_9_12 := FALSE;
    Start_12_9 := FALSE; Start_6_3  := FALSE;
    Start_9_6  := FALSE; Start_3_12 := FALSE;
END_IF


// === Completion check ===
CASE activeRoute OF
    126: IF T12_6_Done THEN Busy := FALSE; activeRoute := 0; END_IF
    612: IF T6_12_Done THEN Busy := FALSE; activeRoute := 0; END_IF
    93 : IF T9_3_Done  THEN Busy := FALSE; activeRoute := 0; END_IF
    39 : IF T3_9_Done  THEN Busy := FALSE; activeRoute := 0; END_IF
    123: IF T12_3_Done THEN Busy := FALSE; activeRoute := 0; END_IF
    69 : IF T6_9_Done  THEN Busy := FALSE; activeRoute := 0; END_IF
    36 : IF T3_6_Done  THEN Busy := FALSE; activeRoute := 0; END_IF
    912: IF T9_12_Done THEN Busy := FALSE; activeRoute := 0; END_IF
    129: IF T12_9_Done THEN Busy := FALSE; activeRoute := 0; END_IF
    63 : IF T6_3_Done  THEN Busy := FALSE; activeRoute := 0; END_IF
    96 : IF T9_6_Done  THEN Busy := FALSE; activeRoute := 0; END_IF
    312: IF T3_12_Done THEN Busy := FALSE; activeRoute := 0; END_IF
END_CASE

METHOD PRIVATE Enqueue : BOOL
VAR_INPUT
    route : INT;
END_VAR

IF QCount < 10 THEN
    queue[tail] := route;
    tail := (tail MOD 10) + 1;
    QCount := QCount + 1;
    Enqueue := TRUE;
ELSE
    Enqueue := FALSE; // queue full
END_IF
END_METHOD

END_FUNCTION_BLOCK

// ---- POUs/FBs/FB_Conveyor.TcPOU
FUNCTION_BLOCK FB_Conveyor
VAR_INPUT
    CmdRunRequest : BOOL;   // scheduler command
    MotorOK       AT%I*: BOOL;   // from sensor
    RunningIn     AT%I*: BOOL;   // from sensor
    PathClear     : BOOL;
END_VAR
VAR_OUTPUT
    MotorRun      AT%Q*: BOOL;   // Output to motor cmd
    IsRunning     : BOOL;
END_VAR
VAR
    Motor : FB_MotorUnit;
END_VAR

Motor(CmdRun := (CmdRunRequest AND PathClear),
      MotorOK := MotorOK,
      RunningIn := RunningIn);

MotorRun  := Motor.MotorRun;
IsRunning := Motor.IsRunning;

END_FUNCTION_BLOCK

// ---- POUs/FBs/FB_Reader.TcPOU
FUNCTION_BLOCK FB_Reader
VAR_INPUT
    TriggerRead : BOOL;   // input from I_ReaderXX_Trigger
	BlueOcc : BOOL;
	ForceDest   : INT := 0; // 0 = random, else fixed destination (12/3/6/9)
	Source : INT;
	Dest : Int;
END_VAR
VAR_OUTPUT
    ReaderValue : INT;    // destination code (12, 3, 6, 9)
    Valid       AT%Q*: BOOL;   // TRUE for one scan when a new value is read
END_VAR
VAR
    lastTrigger : BOOL;
	I_ReaderValue AT%I*:INT;
	vTrigger AT%Q*: BOOL;
    seed        : UDINT := 12345;
    pick        : INT;
END_VAR

// Rising edge detection
IF TriggerRead AND NOT lastTrigger THEN
    IF ForceDest <> 0 THEN
        // Use forced destination
        ReaderValue := ForceDest;
    ELSE
        // Generate random until != Source
        REPEAT
            seed := (1103515245 * seed + 12345);
            CASE (seed MOD 4) OF
                0: pick := 12;
                1: pick := 3;
                2: pick := 6;
                3: pick := 9;
            END_CASE
        UNTIL pick <> Source
        END_REPEAT;
        ReaderValue := pick;
    END_IF
    Valid := TRUE;
ELSE
    Valid := FALSE;
END_IF

lastTrigger := TriggerRead;
//// detect rising edge
//IF TriggerRead AND NOT lastTrigger THEN
//    Valid := TRUE;           // one-cycle pulse
//    ReaderValue := Dest;     // assign destination
//ELSE
//    Valid := FALSE;
//    ReaderValue := 0;
//END_IF

//// update memory
//lastTrigger := TriggerRead;

END_FUNCTION_BLOCK

// ---- POUs/FBs/Interchange/FB_DirectTransferGreen.TcPOU
FUNCTION_BLOCK FB_DirectTransferGreen
VAR_INPUT
    StartRequest : BOOL;   // reader triggered with correct Dest
	JobID        : UDINT;     // unique per dispatch
    LTU1_PosOK   : BOOL;   // e.g. LTU_12_3.PosBottom
    LTU1_Running : BOOL;
    LTU1_LB      : BOOL;   // LightBarrier TRUE=empty
    LTU2_PosOK   : BOOL;   // e.g. LTU_3_6.PosBottom
    LTU2_Running : BOOL;
    LTU2_LB      : BOOL;
    BlueOcc      : BOOL;   // Blue stopper Occupied
END_VAR
VAR_OUTPUT
    BlueCmdDown : BOOL;   // TRUE=block, FALSE=release
	LTU1_MoveDown : BOOL; // True=bottom
	LTU2_MoveDown : BOOL;
	LTU1_MotorRunCmd : BOOL; // True=Run
	LTU2_MotorRunCmd : BOOL;
    Done        : BOOL;
    Error       : BOOL;
END_VAR
VAR
    state    : INT := 0;
    tTimeout : TON;
	reset: BOOL;
	lastRequest: BOOL;
	lastJobID  : UDINT := 0;   // store previous job ID
END_VAR

CASE state OF
0: // IDLE
    BlueCmdDown := TRUE; //Blocking
    Error := FALSE;
	
    // latch Done until new request comes
    IF StartRequest AND JobID <> lastJobID THEN
		// command both LTUs down
        LTU1_MoveDown := TRUE;
        LTU2_MoveDown := TRUE;
        Done := FALSE;        // reset Done on new request
		lastJobID := JobID;
        state := 1;           // start cycle
    END_IF
    

1: // ALIGN
    // keep commanding move down until confirmed
    LTU1_MoveDown := TRUE;
    LTU2_MoveDown := TRUE;

    IF LTU1_PosOK 
       AND LTU2_PosOK  THEN
//        LTU1_MoveDown := FALSE;
//        LTU2_MoveDown := FALSE;
        state := 2; // RELEASE
    END_IF

2: // RELEASE
    IF BlueOcc THEN
        BlueCmdDown := FALSE;   // open for release
        //tTimeout(IN := TRUE, PT := T#8S);
        state := 3;
    END_IF

3: // WAIT_ENTER_LT1
    // Re-block once carrier left Blue
    IF NOT BlueOcc THEN
        BlueCmdDown := TRUE;
    END_IF

    IF NOT LTU1_LB THEN
        state := 4;
//        tTimeout(IN := TRUE, PT := T#8S);
//    ELSIF tTimeout.Q THEN 
//        state := 99; 
    END_IF

4: // WAIT_LEAVE_LT1
	BlueCmdDown := TRUE;//reblock 
	IF LTU1_PosOK 
       AND LTU2_PosOK THEN
		LTU1_MotorRunCmd := TRUE;
		LTU2_MotorRunCmd := TRUE;
	END_IF
    IF LTU1_LB THEN
        state := 5;
//        tTimeout(IN := TRUE, PT := T#8S);
//    ELSIF tTimeout.Q THEN state := 99; 
	END_IF

5: // WAIT_ENTER_LT2
    IF NOT LTU2_LB THEN
        state := 6;
//        tTimeout(IN := TRUE, PT := T#8S);
//    ELSIF tTimeout.Q THEN state := 99; 
	END_IF

6: // WAIT_LEAVE_LT2
    IF LTU2_LB THEN
        BlueCmdDown := TRUE;
        Done := TRUE;
        state := 0;
    //ELSIF tTimeout.Q THEN state := 99; 
	END_IF

99: // ERROR
    BlueCmdDown := TRUE;
    Error := TRUE;
	IF reset THEN
		 state := 0;
	END_IF
   
END_CASE

// --- Edge detection for StartRequest ---
//lastRequest := StartRequest;

END_FUNCTION_BLOCK

// ---- POUs/FBs/Interchange/FB_DirectTransferOrange.TcPOU
FUNCTION_BLOCK FB_DirectTransferOrange
VAR_INPUT
    StartRequest : BOOL;   // reader detected correct dest
	JobID        : UDINT;     // unique per dispatch
    LTU1_PosOK   : BOOL;   // LTU1 at Top
    LTU1_Running : BOOL;
    LTU1_LB      : BOOL;
    LTU2_PosOK   : BOOL;   // LTU2 at Top
    LTU2_Running : BOOL;
    LTU2_LB      : BOOL;
    BlueOcc      : BOOL;   // entry stopper occupied
    Purple1Occ   : BOOL;   // intermediate purple (near LTU1)
    Purple2Occ   : BOOL;   // final purple (exit stopper)
    reset        : BOOL;
END_VAR
VAR_OUTPUT
    BlueCmdDown    : BOOL;
    Purple1CmdDown : BOOL;
    Purple2CmdDown : BOOL;
    LTU1_MoveUp    : BOOL;
    LTU2_MoveUp    : BOOL;
	LTU1_MotorRunCmd : BOOL; // True=bottom
	LTU2_MotorRunCmd : BOOL;
    Done           : BOOL;
    Error          : BOOL;
END_VAR
VAR
    state : INT := 0;
	lastRequest: BOOL;
	lastJobID  : UDINT := 0;   // store previous job ID
END_VAR

CASE state OF
0: // IDLE
    BlueCmdDown    := TRUE;//blocking
    Purple1CmdDown := FALSE;//release
    Purple2CmdDown := FALSE;//release
    Error := FALSE;

    IF StartRequest AND JobID <> lastJobID THEN
        LTU1_MoveUp := TRUE;
        LTU2_MoveUp := TRUE;
		Done := FALSE; 
		lastJobID := JobID;
        state := 1;
    END_IF

1: // ALIGN
    LTU1_MoveUp := TRUE;
    LTU2_MoveUp := TRUE;

    IF LTU1_PosOK AND 
        LTU2_PosOK  THEN
        
        state := 2;
    END_IF

2: // CHECK_PURPLES
    IF (NOT Purple1CmdDown) AND (NOT Purple2CmdDown) THEN
        state := 3;
    END_IF

3: // RELEASE
    IF BlueOcc THEN
        BlueCmdDown := FALSE;
        state := 4;
    END_IF

4: // WAIT_ENTER_LT1
    IF NOT BlueOcc THEN
        BlueCmdDown := TRUE; // re-block entry
    END_IF
	
    IF NOT LTU1_LB THEN
        state := 5;
    END_IF

5: // WAIT_LEAVE_LT1
	BlueCmdDown := TRUE;//reblock 
	LTU1_MotorRunCmd := TRUE;
	LTU2_MotorRunCmd := TRUE;
    IF LTU1_LB THEN
        state := 6;
    END_IF

6: // WAIT_ENTER_LT2
    IF NOT LTU2_LB THEN
        state := 7;
    END_IF

7: // WAIT_LEAVE_LT2
    IF LTU2_LB THEN
        state := 8;
    END_IF

8: // WAIT_AT_PURPLE
    IF Purple2Occ THEN
        Purple2CmdDown := FALSE; // release final carrier
        Done := TRUE;
        state := 0;
    END_IF

99: // ERROR
    BlueCmdDown    := TRUE;
    Purple1CmdDown := TRUE;
    Purple2CmdDown := TRUE;
    Error := TRUE;
    IF reset THEN
        state := 0;
    END_IF
END_CASE

// --- Edge detection for StartRequest ---
lastRequest := StartRequest;

END_FUNCTION_BLOCK

// ---- POUs/FBs/Interchange/FB_TransferCorner_LowerToUpper.TcPOU
FUNCTION_BLOCK FB_TransferCorner_LowerToUpper
VAR_INPUT
    StartRequest : BOOL;   // reader request
	JobID        : UDINT;     // unique per dispatch
    LTU_PosTop   : BOOL;
    LTU_PosBottom: BOOL;
    LTU_Running  : BOOL;   // push motor feedback
    LTU_LB       : BOOL;   // TRUE = empty, FALSE = carrier inside
    BlueOcc      : BOOL;
    PurpleOcc    : BOOL;
    reset        : BOOL;
END_VAR
VAR_OUTPUT
    BlueCmdDown   : BOOL;
    PurpleCmdDown : BOOL;
    LTU_MoveUp    : BOOL;
    LTU_MoveDown  : BOOL;
    LTU_CmdPush   : BOOL;
    Done          : BOOL;
    Error         : BOOL;
END_VAR
VAR
    state : INT := 0;
	lastRequest: BOOL;
	lastJobID  : UDINT := 0;   // store previous job ID
END_VAR

CASE state OF
0: // IDLE
    BlueCmdDown   := TRUE;
    PurpleCmdDown := TRUE;
    LTU_MoveUp    := FALSE;
    LTU_MoveDown  := TRUE;   // stay aligned to Bottom by default
    LTU_CmdPush   := FALSE;
    Error := FALSE;

    // latch Done until a new StartRequest arrives
    IF StartRequest AND JobID <> lastJobID THEN
        Done := FALSE;           // clear done on new request
		lastJobID := JobID;
        state := 1;              // start new transfer
    END_IF

1: // RELEASE BLUE
    IF BlueOcc AND LTU_PosBottom THEN
        BlueCmdDown := FALSE;   // let carrier enter LTU
        state := 2;
    END_IF

2: // WAIT ENTER LTU
    IF NOT BlueOcc THEN
        BlueCmdDown := TRUE;    // re-block entry
    END_IF
    IF NOT LTU_LB THEN          // LTU occupied
        state := 3;
    END_IF

3: // LIFT TO TOP
	BlueCmdDown := TRUE;
    LTU_MoveDown := FALSE;
    LTU_MoveUp   := TRUE;

    IF LTU_PosTop THEN
        LTU_MoveUp := FALSE;
        state := 4;
    END_IF

4: // PUSH OUT
    IF PurpleOcc THEN
        PurpleCmdDown := FALSE;
    END_IF
     
    IF NOT PurpleCmdDown THEN   // only push if exit released
        LTU_CmdPush := TRUE;
        IF PurpleOcc THEN
            LTU_CmdPush := FALSE;
            Done := TRUE;      // latch Done here
            state := 0;        // return to IDLE, but Done stays TRUE
        END_IF
    END_IF

99: // ERROR
    BlueCmdDown   := TRUE;
    PurpleCmdDown := TRUE;
    LTU_MoveUp    := FALSE;
    LTU_MoveDown  := FALSE;
    LTU_CmdPush   := FALSE;
    Error := TRUE;
    IF reset THEN
        state := 0;
    END_IF
END_CASE

// Rising edge detector for StartRequest
lastRequest := StartRequest;

END_FUNCTION_BLOCK

// ---- POUs/FBs/Interchange/FB_TransferCorner_UpperToLower.TcPOU
FUNCTION_BLOCK FB_TransferCorner_UpperToLower
VAR_INPUT
    StartRequest : BOOL;   // request to start
	JobID        : UDINT;     // unique per dispatch
    LTU_PosTop   : BOOL;
    LTU_PosBottom: BOOL;
    LTU_Running  : BOOL;
    LTU_LB       : BOOL;   // TRUE=empty, FALSE=occupied
    BlueOcc      : BOOL;   // Blue entry occupied
    PurpleOcc    : BOOL;   // entry purple occupied (must be released)
    reset        : BOOL;
END_VAR
VAR_OUTPUT
    BlueCmdDown   : BOOL;
    PurpleCmdDown : BOOL;
    LTU_MoveUp    : BOOL;
    LTU_MoveDown  : BOOL;
    LTU_CmdPush   : BOOL;
    Done          : BOOL;
    Error         : BOOL;
END_VAR
VAR
    state : INT := 0;
	lastRequest: BOOL;
	lastJobID  : UDINT := 0;   // store previous job ID
END_VAR

CASE state OF
0: // IDLE
    BlueCmdDown   := TRUE;
    PurpleCmdDown := TRUE;   // block by default
    LTU_MoveUp    := TRUE;   // keep aligned to Top
    LTU_MoveDown  := FALSE;
    LTU_CmdPush   := FALSE;
    Error := FALSE;

    // latch Done until new request comes
    IF StartRequest AND JobID <> lastJobID THEN
        Done := FALSE;        // reset Done on new request
		lastJobID := JobID;
        state := 1;           // start cycle
    END_IF

1: // ALIGN TOP
    LTU_MoveUp := TRUE;
    IF LTU_PosTop AND NOT LTU_Running THEN
        LTU_MoveUp := FALSE;
        state := 2;
    END_IF

2: // RELEASE
    IF BlueOcc AND PurpleCmdDown THEN
        BlueCmdDown := FALSE;  // let carrier into LTU
        state := 3;
    END_IF

3: // WAIT_ENTER_LT
    IF NOT BlueOcc THEN
        BlueCmdDown := TRUE;   // re-block entry
    END_IF
    IF NOT LTU_LB THEN
        state := 4;
    END_IF

4: // LIFT DOWN
	BlueCmdDown := TRUE;//reblock 
    LTU_MoveDown := TRUE;
    IF LTU_PosBottom AND NOT LTU_Running THEN
        LTU_MoveDown := FALSE;
        state := 5;
    END_IF

5: // PUSH OUT
    LTU_CmdPush := TRUE;
    IF LTU_LB THEN  // became empty again
        LTU_CmdPush := FALSE;
        Done := TRUE;         // latch Done
        state := 0;           // go back to IDLE
    END_IF

99: // ERROR
    BlueCmdDown   := TRUE;
    PurpleCmdDown := TRUE;
    LTU_MoveUp    := FALSE;
    LTU_MoveDown  := FALSE;
    LTU_CmdPush   := FALSE;
    Error := TRUE;
    IF reset THEN
        state := 0;
    END_IF
END_CASE

// --- Edge detection for StartRequest ---
lastRequest := StartRequest;

END_FUNCTION_BLOCK

// ---- POUs/FBs/Interchange/FB_TransferChain_LowerToUpper.TcPOU
FUNCTION_BLOCK FB_TransferChain_LowerToUpper
VAR_INPUT
    StartRequest : BOOL;
	JobID        : UDINT;     // unique per dispatch
    reset        : BOOL;

    // Blue12
    BlueOcc      : BOOL;

    // LTU_12_3
    LTU1_PosBottom, LTU1_PosTop, LTU1_Running, LTU1_LB : BOOL;

    // LTU_3_6
    LTU2_PosBottom, LTU2_PosTop, LTU2_Running, LTU2_LB : BOOL;

    // LTU_6_9
    LTU3_PosBottom, LTU3_PosTop, LTU3_Running, LTU3_LB : BOOL;

    // Purple stoppers
    Purple1_Occ : BOOL;   // Purple9_3_2
    Purple2_Occ : BOOL;   // Purple3_9_1
    Purple3_Occ : BOOL;   // Purple3_9_2
END_VAR
VAR_OUTPUT
    // Blue
    BlueCmdDown : BOOL;

    // Purple
    Purple1CmdDown, Purple2CmdDown, Purple3CmdDown : BOOL;

    // LTU_12_3
    LTU1_CmdPush, LTU1_MoveUp, LTU1_MoveDown : BOOL;

    // LTU_3_6
    LTU2_CmdPush, LTU2_MoveUp, LTU2_MoveDown : BOOL;

    // LTU_6_9
    LTU3_CmdPush, LTU3_MoveUp, LTU3_MoveDown : BOOL;

    Done  : BOOL;
    Error : BOOL;
END_VAR
VAR
    state       : INT := 0;
    lastRequest : BOOL := FALSE;
	lastJobID  : UDINT := 0;   // store previous job ID
END_VAR

CASE state OF
0: // IDLE
    BlueCmdDown     := TRUE;
    Purple1CmdDown  := TRUE;
    Purple2CmdDown  := TRUE;
    Purple3CmdDown  := TRUE;
	LTU1_MoveDown := FALSE;
	LTU1_MoveUp := FALSE;
	LTU2_MoveDown := FALSE;
	LTU2_MoveUp := FALSE;
	LTU3_MoveDown := FALSE;
	LTU3_MoveUp := FALSE;
	
	
    LTU1_CmdPush := FALSE;
    LTU2_CmdPush := FALSE;
    LTU3_CmdPush := FALSE;

    Error := FALSE;

    IF StartRequest AND JobID <> lastJobID THEN
        Done := FALSE;
		lastJobID := JobID;
        state := 1;
    END_IF

1: // ALIGN
    LTU1_MoveDown := TRUE;   // LTU_12_3 to Bottom
    LTU2_MoveDown := TRUE;   // LTU_3_6 to Bottom
    LTU3_MoveUp   := TRUE;   // LTU_6_9 to Top

    IF LTU1_PosBottom AND NOT LTU1_Running
       AND LTU2_PosBottom AND NOT LTU2_Running
       AND LTU3_PosTop AND NOT LTU3_Running THEN
        state := 2;
    END_IF

2: // CHECK_PURPLES
    IF Purple1CmdDown AND Purple2CmdDown AND Purple3CmdDown THEN
        state := 3;
    END_IF

3: // RELEASE BLUE
    IF BlueOcc THEN
        BlueCmdDown := FALSE;
        state := 4;
    END_IF

4: // LTU_12_3 cycle (straight push to LTU_3_6)
    IF NOT BlueOcc THEN 
		BlueCmdDown := TRUE; //reblocking after release
	END_IF

    IF NOT LTU1_LB AND NOT LTU2_Running THEN //carrier reached LTU1 and LTU2 is not running
        LTU1_CmdPush := TRUE;
    END_IF

    IF LTU1_LB THEN
        LTU1_CmdPush := FALSE;
        state := 5;
    END_IF

5: // LTU_3_6 cycle (Lift Up + Push to Purple3_9_1)
	BlueCmdDown := TRUE; //reblocking after release
    IF NOT LTU2_LB THEN //carrier reached LTU2
        LTU2_MoveUp := TRUE;
		LTU2_MoveDown := FALSE;
        IF LTU2_PosTop AND NOT LTU3_Running THEN
            //LTU2_MoveUp := FALSE;
            LTU2_CmdPush := TRUE;
            IF Purple2_Occ THEN
                //LTU2_CmdPush := FALSE;
                state := 6;
            END_IF
        END_IF
    END_IF

6: // RELEASE Purple3_9_1
    Purple2CmdDown := FALSE;
	IF NOT Purple2_Occ THEN
		LTU2_CmdPush := FALSE;
		state := 7;
	END_IF
    

7: // LTU_6_9 cycle (Bottom->Top->Push to Purple9_3_2)
    IF NOT LTU3_LB THEN// carrier is reached LTU3
        LTU3_MoveUp := TRUE;
		LTU3_MoveDown := FALSE;
        IF LTU3_PosTop  THEN
            //LTU3_MoveUp := FALSE;
            LTU3_CmdPush := TRUE;
            IF Purple3_Occ THEN
                //LTU3_CmdPush := FALSE;
                state := 8;
            END_IF
        END_IF
    END_IF

8: // COMPLETE
    Purple3CmdDown := FALSE;
	IF NOT Purple3_Occ THEN
		LTU3_CmdPush := FALSE;
		Done := TRUE;
    	state := 0;
	END_IF
 

99: // ERROR
    BlueCmdDown     := TRUE;
    Purple1CmdDown  := TRUE;
    Purple2CmdDown  := TRUE;
    Purple3CmdDown  := TRUE;
    LTU1_CmdPush := FALSE;
    LTU2_CmdPush := FALSE;
    LTU3_CmdPush := FALSE;
    Error := TRUE;
    IF reset THEN state := 0; END_IF
END_CASE

// latch new request
lastRequest := StartRequest;

END_FUNCTION_BLOCK

// ---- POUs/FBs/Interchange/FB_TransferChain_UpperToLower.TcPOU
FUNCTION_BLOCK FB_TransferChain_UpperToLower
VAR_INPUT
    StartRequest : BOOL;
	JobID        : UDINT;     // unique per dispatch
    reset        : BOOL;

    // Blue9
    BlueOcc      : BOOL;

    // LTU_9_12
    LTU1_PosBottom, LTU1_PosTop, LTU1_Running, LTU1_LB : BOOL;

    // LTU_12_3
    LTU2_PosBottom, LTU2_PosTop, LTU2_Running, LTU2_LB : BOOL;

    // LTU_3_6
    LTU3_PosBottom, LTU3_PosTop, LTU3_Running, LTU3_LB : BOOL;

    // Purple stoppers
    Purple1_Occ : BOOL;   // Purple9_3_1
    Purple2_Occ : BOOL;   // Purple9_3_2
	Purple3_Occ : BOOL;   // Purple3_9_1
END_VAR
VAR_OUTPUT
    BlueCmdDown : BOOL;

    Purple1CmdDown, Purple2CmdDown, Purple3CmdDown : BOOL;

    // LTU_9_12
    LTU1_CmdPush, LTU1_MoveUp, LTU1_MoveDown : BOOL;

    // LTU_12_3
    LTU2_CmdPush, LTU2_MoveUp, LTU2_MoveDown : BOOL;

    // LTU_3_6
    LTU3_CmdPush, LTU3_MoveUp, LTU3_MoveDown : BOOL;

    Done  : BOOL;
    Error : BOOL;
END_VAR
VAR
    state       : INT := 0;
    lastRequest : BOOL := FALSE;
	lastJobID  : UDINT := 0;   // store previous job ID
END_VAR

CASE state OF
0: // IDLE
    BlueCmdDown     := TRUE;
    Purple1CmdDown  := TRUE;
    Purple2CmdDown  := TRUE;

    LTU1_CmdPush := FALSE;
    LTU2_CmdPush := FALSE;
    LTU3_CmdPush := FALSE;

    LTU1_MoveUp := FALSE; LTU1_MoveDown := FALSE;
    LTU2_MoveUp := FALSE; LTU2_MoveDown := FALSE;
    LTU3_MoveUp := FALSE; LTU3_MoveDown := FALSE;

    Error := FALSE;

    IF StartRequest AND JobID <> lastJobID THEN
        Done := FALSE;
		lastJobID := JobID;
        state := 1;
    END_IF

1: // ALIGN
    LTU1_MoveUp   := TRUE;   // LTU_9_12 to Top
    LTU2_MoveUp   := TRUE;   // LTU_12_3 to Top
    LTU3_MoveDown := TRUE;   // LTU_3_6 to Bottom

    IF LTU1_PosTop AND NOT LTU1_Running
       AND LTU2_PosTop AND NOT LTU2_Running
       AND LTU3_PosBottom AND NOT LTU3_Running THEN
        LTU1_MoveUp   := FALSE;
        LTU2_MoveUp   := FALSE;
        LTU3_MoveDown := FALSE;
        state := 2;
    END_IF

2: // CHECK_PURPLES
    IF Purple1CmdDown AND Purple2CmdDown THEN
        state := 3;
    END_IF

3: // RELEASE BLUE9
    IF BlueOcc THEN
        BlueCmdDown := FALSE;
        state := 4;
    END_IF

4: // LTU_9_12 push
    IF NOT BlueOcc THEN 
		BlueCmdDown := TRUE;//reblock 
	END_IF

    IF NOT LTU1_LB THEN
        LTU1_CmdPush := TRUE;
    END_IF

    IF LTU1_LB THEN
        LTU1_CmdPush := FALSE;
        state := 5;
    END_IF

5: // RELEASE Purple9_3_1
	BlueCmdDown := TRUE;//reblock 
    Purple1CmdDown := FALSE;
    IF NOT Purple1_Occ THEN
        state := 6;
    END_IF

6: // LTU_12_3 cycle (Down + Push)
    IF NOT LTU2_LB THEN//carrier is reached LTU2 
        LTU2_MoveDown := TRUE;
        IF LTU2_PosBottom AND NOT LTU3_Running THEN
            //LTU2_MoveDown := FALSE;
            LTU2_CmdPush := TRUE;
            state := 7;
        END_IF
    END_IF

//7: // RELEASE Purple9_3_2
//    Purple2CmdDown := FALSE;
//    IF NOT Purple2_Occ THEN
//        state := 8;
//    END_IF

7: // LTU_3_6 push (already at Bottom)
	IF LTU2_LB THEN
		LTU2_CmdPush := FALSE;
	END_IF
    IF NOT LTU3_LB THEN
        LTU3_CmdPush := TRUE;
    END_IF
	IF LTU3_LB THEN
		LTU3_CmdPush := FALSE;
		Done := TRUE;
		state := 0;
	END_IF

99: // ERROR
    BlueCmdDown     := TRUE;
    Purple1CmdDown  := TRUE;
    Purple2CmdDown  := TRUE;
    LTU1_CmdPush := FALSE;
    LTU2_CmdPush := FALSE;
    LTU3_CmdPush := FALSE;
    Error := TRUE;
    IF reset THEN state := 0; END_IF
END_CASE

// latch new request
lastRequest := StartRequest;

END_FUNCTION_BLOCK

// ---- POUs/FBs/Scheduler/FB_ThroughputMonitor.TcPOU
FUNCTION_BLOCK FB_ThroughputMonitor
VAR_INPUT
    DonePulse : BOOL;     // one-scan TRUE when a transfer completes
    Reset     : BOOL;     // reset counters
END_VAR
VAR_OUTPUT
    TotalCount        : UDINT;   // total carriers processed
    PerMinute         : UDINT;   // carriers per minute
    PerHour           : UDINT;   // carriers per hour
    LastSampleCount   : UDINT;   // carriers seen in last sample window
END_VAR
VAR
    tSample   : TON;      // 1-minute sampling timer
    prevDone  : BOOL;
    lastTotal : UDINT;
END_VAR

// --- Reset logic ---
IF Reset THEN
    TotalCount := 0;
    PerMinute := 0;
    PerHour := 0;
    LastSampleCount := 0;
    lastTotal := 0;
END_IF


// --- Count Done pulses ---
IF DonePulse AND NOT prevDone THEN
    TotalCount := TotalCount + 1;
END_IF
prevDone := DonePulse;


// --- Run 60s timer ---
tSample(IN := TRUE, PT := T#60s);

// When timer completes → sample throughput
IF tSample.Q THEN
    LastSampleCount := TotalCount - lastTotal; // carriers in last 60s
    PerMinute := LastSampleCount;
    PerHour   := LastSampleCount * 60;
    lastTotal := TotalCount;

    // restart timer
    tSample(IN := FALSE);
END_IF

END_FUNCTION_BLOCK

// ---- POUs/FBs/Homing/FB_HomingManager.TcPOU
FUNCTION_BLOCK FB_HomingManager
VAR_INPUT
    StartHoming : BOOL;
    Reset       : BOOL;

    // LTU inputs
    LTU_12_3_PosTop, LTU_12_3_PosBottom, LTU_12_3_PosMid, LTU_12_3_Running : BOOL;
    LTU_3_6_PosTop, LTU_3_6_PosBottom, LTU_3_6_PosMid, LTU_3_6_Running     : BOOL;
    LTU_9_12_PosTop, LTU_9_12_PosBottom, LTU_9_12_PosMid, LTU_9_12_Running : BOOL;
    LTU_6_9_PosTop, LTU_6_9_PosBottom, LTU_6_9_PosMid, LTU_6_9_Running     : BOOL;
END_VAR
VAR_OUTPUT
    LTU_12_3_CmdMoveUp, LTU_12_3_CmdMoveDown : BOOL;
    LTU_3_6_CmdMoveUp,  LTU_3_6_CmdMoveDown  : BOOL;
    LTU_9_12_CmdMoveUp, LTU_9_12_CmdMoveDown : BOOL;
    LTU_6_9_CmdMoveUp,  LTU_6_9_CmdMoveDown  : BOOL;

    AllDone   : BOOL;
    AnyError  : BOOL;
END_VAR
VAR
    Home_12_3 : FB_HomingLTU;
    Home_3_6  : FB_HomingLTU;
    Home_9_12 : FB_HomingLTU;
    Home_6_9  : FB_HomingLTU;
END_VAR

// --- Run all homing FBs in parallel ---
Home_12_3(
    StartHoming := StartHoming,
    Reset       := Reset,
    PosTop      := LTU_12_3_PosTop,
    PosBottom   := LTU_12_3_PosBottom,
    PosMid      := LTU_12_3_PosMid,
    Running     := LTU_12_3_Running,
    CmdMoveDown => LTU_12_3_CmdMoveDown,
    CmdMoveUp   => LTU_12_3_CmdMoveUp
);

Home_3_6(
    StartHoming := StartHoming,
    Reset       := Reset,
    PosTop      := LTU_3_6_PosTop,
    PosBottom   := LTU_3_6_PosBottom,
    PosMid      := LTU_3_6_PosMid,
    Running     := LTU_3_6_Running,
    CmdMoveDown => LTU_3_6_CmdMoveDown,
    CmdMoveUp   => LTU_3_6_CmdMoveUp
);

Home_9_12(
    StartHoming := StartHoming,
    Reset       := Reset,
    PosTop      := LTU_9_12_PosTop,
    PosBottom   := LTU_9_12_PosBottom,
    PosMid      := LTU_9_12_PosMid,
    Running     := LTU_9_12_Running,
    CmdMoveDown => LTU_9_12_CmdMoveDown,
    CmdMoveUp   => LTU_9_12_CmdMoveUp
);

Home_6_9(
    StartHoming := StartHoming,
    Reset       := Reset,
    PosTop      := LTU_6_9_PosTop,
    PosBottom   := LTU_6_9_PosBottom,
    PosMid      := LTU_6_9_PosMid,
    Running     := LTU_6_9_Running,
    CmdMoveDown => LTU_6_9_CmdMoveDown,
    CmdMoveUp   => LTU_6_9_CmdMoveUp
);


// --- Manager Outputs ---
AllDone  := Home_12_3.Done AND Home_3_6.Done AND Home_9_12.Done AND Home_6_9.Done;
AnyError := Home_12_3.Error OR Home_3_6.Error OR Home_9_12.Error OR Home_6_9.Error;

END_FUNCTION_BLOCK

// ---- POUs/FBs/Homing/FB_HomingLTU.TcPOU
FUNCTION_BLOCK FB_HomingLTU
VAR_INPUT
    StartHoming : BOOL;
    Reset       : BOOL;

    PosTop      : BOOL;
    PosBottom   : BOOL;
    PosMid      : BOOL;
    Running     : BOOL;
END_VAR
VAR_OUTPUT
    CmdMoveDown : BOOL;
    CmdMoveUp   : BOOL;
    Done        : BOOL;
    Error       : BOOL;
END_VAR
VAR
    state       : INT := 0;
    tTimeout    : TON;
END_VAR

CASE state OF
    0: // IDLE
        CmdMoveDown := FALSE;
        CmdMoveUp   := FALSE;
        Done  := FALSE;
        Error := FALSE;

        IF StartHoming THEN
            state := 1;
        END_IF

    1: // MOVE DOWN
        CmdMoveDown := TRUE;
        CmdMoveUp   := FALSE;

        tTimeout(IN:=TRUE, PT:=T#10s);

        IF PosBottom THEN
            CmdMoveDown := FALSE;
            Done := TRUE;
            tTimeout(IN:=FALSE);
            state := 2;
        ELSIF tTimeout.Q THEN
            Error := TRUE;
            CmdMoveDown := FALSE;
            state := 99;
        END_IF

    2: // HOMED
        // Hold here until reset
        CmdMoveDown := FALSE;
        CmdMoveUp   := FALSE;
        Done := TRUE;
        IF Reset THEN
            state := 0;
        END_IF

    99: // ERROR
        CmdMoveDown := FALSE;
        CmdMoveUp   := FALSE;
        Error := TRUE;
        IF Reset THEN
            state := 0;
        END_IF
END_CASE

END_FUNCTION_BLOCK

// ---- POUs/FCs/FB_AutoPlace.TcPOU
FUNCTION_BLOCK FB_AutoPlace
VAR_INPUT
	BlueStopper : BOOL;
	
END_VAR
VAR_OUTPUT
	Reader_Trigger : BOOL;
END_VAR
VAR
	Cont_Timer : ton;
	last_triggered: BOOL;
	start: BOOL;
END_VAR


Cont_Timer(IN:= BlueStopper, PT:= T#3S, Q=> , ET=> );
IF BlueStopper AND Cont_Timer.Q THEN
	//
	Reader_Trigger := TRUE;
ELSE 
	//
	Reader_Trigger := FALSE;
END_IF

//last_triggered := BlueStopper;

END_FUNCTION_BLOCK

// ---- POUs/PRG_SIM.TcPOU
PROGRAM PRG_SIM
VAR
 SimConv12_6 : FB_SimConveyor;
 SimConv6_12 : FB_SimConveyor;
 SimConv3_9 : FB_SimConveyor;
 SimConv9_3 : FB_SimConveyor;

 SimBlue12 : FB_SimStopper;
 SimBlue6 : FB_SimStopper;
 SimBlue3 : FB_SimStopper;
 SimBlue9 : FB_SimStopper;
 
 SimLTU12_3 : FB_SimLTU;
 SimLTU3_6 : FB_SimLTU;
 SimLTU6_9 : FB_SimLTU;
 SimLTU9_12 : FB_SimLTU;
 
 SimPurp9_3_1: FB_SimStopper;
 SimPurp9_3_2 : FB_SimStopper;
 SimPurp3_9_1: FB_SimStopper;
 SimPurp3_9_2 : FB_SimStopper;
 
 SimReader_12 : FB_SimReader;
 SimReader_3 : FB_SimReader;
 SimReader_6 : FB_SimReader;
 SimReader_9 : FB_SimReader;
 
 Inject_12_3 : FB_InjectAfterRelease;
 Inject_3_6  : FB_InjectAfterRelease;
 Inject_12_9 : FB_InjectAfterRelease;
 Inject_9_6  : FB_InjectAfterRelease;
 Inject_Trial  : FB_InjectAfterRelease;

 prevBlue12Occ, prevBlue3Occ, prevBlue6Occ, prevBlue9Occ : BOOL;
 
 LTU_12_3_CarrierIn : BOOL;
 LTU_3_6_CarrierIn : BOOL;
 LTU_12_9_CarrierIn : BOOL;
 LTU_9_6_CarrierIn : BOOL;
	ReleaseTrig: BOOL;
	CarrierIn: BOOL;
END_VAR

SimConv12_6(
	MotorRun:= , 
	Release:= , 
	MotorOK=> , 
	RunningIn=> , 
	CarrierAtIn=> , 
	CarrierAtOut=> );

SimConv6_12(
	MotorRun:= , 
	Release:= , 
	MotorOK=> , 
	RunningIn=> , 
	CarrierAtIn=> , 
	CarrierAtOut=> );
	
SimConv3_9(
	MotorRun:= , 
	Release:= , 
	MotorOK=> , 
	RunningIn=> , 
	CarrierAtIn=> , 
	CarrierAtOut=> );
	
SimConv9_3(
	MotorRun:= , 
	Release:= , 
	MotorOK=> , 
	RunningIn=> , 
	CarrierAtIn=> , 
	CarrierAtOut=> );
	
SimReader_12(
	TriggerRead:= , 
	ForceDest:= 6, 
	Source:= 12, 
	ReaderValue=> , 
	Valid=> );
SimReader_3(
	TriggerRead:= , 
	ForceDest:= 0, 
	Source:= 3, 
	ReaderValue=> , 
	Valid=> );
SimReader_6(
	TriggerRead:= , 
	ForceDest:= 0, 
	Source:= 6, 
	ReaderValue=> , 
	Valid=> );
SimReader_9(
	TriggerRead:= , 
	ForceDest:= 0, 
	Source:= 9, 
	ReaderValue=> , 
	Valid=> );		
	
SimBlue12(CmdDown:= , CarrierIn:= , Occupied=> , CarrierOut=> );
SimBlue6(CmdDown:= , CarrierIn:= , Occupied=> , CarrierOut=> );
SimBlue3(CmdDown:= , CarrierIn:= , Occupied=> , CarrierOut=> );
SimBlue9(CmdDown:= , CarrierIn:= , Occupied=> , CarrierOut=> );

SimPurp9_3_1(CmdDown:= , CarrierIn:= , Occupied=> , CarrierOut=> );
SimPurp9_3_2(CmdDown:= , CarrierIn:= , Occupied=> , CarrierOut=> );
SimPurp3_9_1(CmdDown:= , CarrierIn:= , Occupied=> , CarrierOut=> );
SimPurp3_9_2(CmdDown:= , CarrierIn:= , Occupied=> , CarrierOut=> );


SimLTU12_3(
	CmdPush:= , 
	MoveUp:= , 
	MoveDown:= , 
	CarrierIn:= , 
	MotorOK=> , 
	PushRunning=> , 
	PosTop=> , 
	PosMid=> , 
	PosBottom=> , 
	LightBarrier=> , 
	CarrierOut=> , 
	Occupied=> , 
	LiftBusy=> );
	
SimLTU3_6(
	CmdPush:= , 
	MoveUp:= , 
	MoveDown:= , 
	CarrierIn:= , 
	MotorOK=> , 
	PushRunning=> , 
	PosTop=> , 
	PosMid=> , 
	PosBottom=> , 
	LightBarrier=> , 
	CarrierOut=> , 
	Occupied=> , 
	LiftBusy=> );
	
SimLTU6_9(
	CmdPush:= , 
	MoveUp:= , 
	MoveDown:= , 
	CarrierIn:= , 
	MotorOK=> , 
	PushRunning=> , 
	PosTop=> , 
	PosMid=> , 
	PosBottom=> , 
	LightBarrier=> , 
	CarrierOut=> , 
	Occupied=> , 
	LiftBusy=> );
	
SimLTU9_12(
	CmdPush:= , 
	MoveUp:= , 
	MoveDown:= , 
	CarrierIn:= LTU_12_9_CarrierIn, 
	MotorOK=> , 
	PushRunning=> , 
	PosTop=> , 
	PosMid=> , 
	PosBottom=> , 
	LightBarrier=> , 
	CarrierOut=> , 
	Occupied=> , 
	LiftBusy=> );

END_PROGRAM

// ---- POUs/Simulation/FB_SimConveyor.TcPOU
FUNCTION_BLOCK FB_SimConveyor
VAR_INPUT
    MotorRun AT%I*: BOOL;   // from MAIN
    Release  AT%I*: BOOL;   // TRUE = stopper released
END_VAR
VAR_OUTPUT
    MotorOK     AT%Q*: BOOL;   // always TRUE in sim
    RunningIn   AT%Q*: BOOL;   // motor feedback
    CarrierAtIn : BOOL;   // entry sensor
    CarrierAtOut: BOOL;   // exit sensor
END_VAR
VAR
    tRun : TON;
    CarrierPresent : BOOL := TRUE;  // assume one carrier available at start
    TravelTime     : TIME := T#3S;
END_VAR


MotorOK   := TRUE;
RunningIn := MotorRun;

// Start travel timer if conveyor runs and release open
tRun(IN := MotorRun AND Release AND CarrierPresent, PT := TravelTime);

// Entry sensor active while carrier present
CarrierAtIn := CarrierPresent;

// When travel done → move carrier to exit
IF CarrierPresent AND tRun.Q THEN
    CarrierAtIn  := FALSE;
    CarrierAtOut := TRUE;
    CarrierPresent := FALSE;
END_IF

END_FUNCTION_BLOCK

// ---- POUs/Simulation/FB_SimStopper.TcPOU
FUNCTION_BLOCK FB_SimStopper
VAR_INPUT
    CmdDown    AT%I*: BOOL;   // from MAIN: TRUE=block, FALSE=release
    CarrierIn  at%I*: BOOL;   // simulated incoming carrier (from conveyor or LTU)
END_VAR
VAR_OUTPUT
    Occupied   AT%Q*: BOOL;   // TRUE when carrier is latched at stopper
    CarrierOut : BOOL;   // TRUE when carrier passes through
END_VAR
VAR
    Latched : BOOL;
END_VAR



// Latch carrier if stopper is down and one arrives
IF CarrierIn AND CmdDown THEN
    Latched := TRUE;
END_IF

// Release carrier if stopper is up
IF NOT CmdDown AND Latched THEN
    Latched := FALSE;
    CarrierOut := TRUE;      // carrier moves forward
ELSE
    CarrierOut := FALSE;     // default
END_IF

// Occupied means stopper currently holding a carrier
Occupied := Latched;

END_FUNCTION_BLOCK

// ---- POUs/Simulation/FB_SimLTU.TcPOU
FUNCTION_BLOCK FB_SimLTU
VAR_INPUT
    CmdPush   AT%I*: BOOL;   // push motor command from MAIN (O_LTU_xx_MotorRun)
    MoveUp    AT%I*: BOOL;   // lift up (hold to continue stepping up)
    MoveDown  AT%I*: BOOL;   // lift down (hold to continue stepping down)
    CarrierIn : BOOL;   // carrier entering LTU from conveyor/stopper
END_VAR
VAR_OUTPUT
    MotorOK     AT%Q*: BOOL;   // always TRUE in sim
    PushRunning AT%Q*: BOOL;   // push motor feedback (RunningIn)
    PosTop      AT%Q*: BOOL;   // LTU aligned with orange/top
    PosMid      AT%Q*: BOOL;   // LTU at middle stop
    PosBottom   AT%Q*: BOOL;   // LTU aligned with green/bottom
    LightBarrier AT%Q*: BOOL;   // TRUE = empty, FALSE = carrier inside
    CarrierOut  : BOOL;   // TRUE for one scan when carrier pushed out
    Occupied    : BOOL;   // TRUE when LTU holds a carrier
    LiftBusy    : BOOL;   // TRUE while lift is moving
	Error       : BOOL;   // TRUE if invalid outputs
END_VAR
VAR
    tUp, tDown  : TON;
    tPush       : TON;
    CarrierInside: BOOL;
END_VAR

// === Motor always healthy ===
MotorOK := TRUE;
PushRunning := CmdPush;

// === Truth table for lift ===
IF (MoveDown AND MoveUp) THEN
    Error := TRUE; // invalid condition
ELSIF MoveDown THEN
    PosBottom := TRUE;
    PosMid    := FALSE;
    PosTop    := FALSE;
    LiftBusy  := TRUE;
    Error     := FALSE;
ELSIF MoveUp THEN
    PosBottom := FALSE;
    PosMid    := FALSE;
    PosTop    := TRUE;
    LiftBusy  := TRUE;
    Error     := FALSE;
ELSE
    PosBottom := FALSE;
    PosMid    := TRUE;
    PosTop    := FALSE;
    LiftBusy  := FALSE;
    Error     := FALSE;
END_IF

// === Carrier entering LTU (handshake) ===
IF CarrierIn AND NOT CarrierInside THEN
    CarrierInside := TRUE;
    CarrierIn := FALSE; // consume the carrier from injector
END_IF

// Light barrier & occupancy
LightBarrier := NOT CarrierInside;
Occupied     := CarrierInside;

// === Push motor simulation ===
tPush(IN := CmdPush AND CarrierInside, PT := T#2S);

IF CarrierInside AND tPush.Q THEN
    CarrierInside := FALSE;  // carrier leaves LTU
    CarrierOut    := TRUE;   // one-cycle pulse
ELSE
    CarrierOut := FALSE;
END_IF

END_FUNCTION_BLOCK

// ---- POUs/Simulation/FB_SimReader.TcPOU
FUNCTION_BLOCK FB_SimReader
VAR_INPUT
    TriggerRead AT%I*: BOOL;   // pulse from simulation (like tTrig.Q)
    ForceDest   : INT := 0; // 0 = random, else fixed destination (12/3/6/9)
	Source      : INT;      // reader's location (12,3,6,9)
END_VAR
VAR_OUTPUT
    ReaderValue AT%Q*: INT;    // chosen destination
    Valid       : BOOL;   // TRUE for one cycle
END_VAR
VAR
    lastTrigger : BOOL;
    seed        : UDINT := 12345;
    pick        : INT;
END_VAR

// Rising edge detection
IF TriggerRead AND NOT lastTrigger THEN
    IF ForceDest <> 0 THEN
        // Use forced destination
        ReaderValue := ForceDest;
    ELSE
        // Generate random until != Source
        REPEAT
            seed := (1103515245 * seed + 12345);
            CASE (seed MOD 4) OF
                0: pick := 12;
                1: pick := 3;
                2: pick := 6;
                3: pick := 9;
            END_CASE
        UNTIL pick <> Source
        END_REPEAT;
        ReaderValue := pick;
    END_IF
    Valid := TRUE;
ELSE
    Valid := FALSE;
END_IF

lastTrigger := TriggerRead;

END_FUNCTION_BLOCK

// ---- POUs/Simulation/FB_InjectAfterRelease.TcPOU
FUNCTION_BLOCK FB_InjectAfterRelease
VAR_INPUT
    ReleaseTrig : BOOL;    // e.g. Blue stop occupied -> free
    PT_Travel   : TIME;    // travel time
END_VAR
VAR_OUTPUT
    CarrierIn   : BOOL;    // pulse
END_VAR
VAR
    tTravel   : TON;
    prevTrig  : BOOL;
    travelDone: BOOL;
END_VAR

// Detect falling edge of ReleaseTrig
IF ReleaseTrig AND NOT prevTrig THEN
    tTravel(IN := TRUE, PT := PT_Travel);
    travelDone := FALSE;
END_IF

// Timer completes → latch CarrierIn
IF tTravel.Q THEN
    CarrierIn := TRUE;
    travelDone := TRUE;
    tTravel(IN := FALSE);
END_IF

// Once LTU consumes the carrier, its SimLTU will reset CarrierIn → FALSE
IF NOT travelDone THEN
    CarrierIn := FALSE;
END_IF

// Save trigger state
prevTrig := ReleaseTrig;

END_FUNCTION_BLOCK

// ---- POUs/FBs/Scheduler/FB_Scheduler.TcPOU
FUNCTION_BLOCK FB_Scheduler
VAR_INPUT
    // Reader inputs
    Reader12_Valid : BOOL;
    Reader12_Value : INT;

    Reader3_Valid  : BOOL;
    Reader3_Value  : INT;

    Reader6_Valid  : BOOL;
    Reader6_Value  : INT;

    Reader9_Valid  : BOOL;
    Reader9_Value  : INT;

    // Transfer Done flags (from all FBs)
    T12_6_Done, T6_12_Done : BOOL;
    T9_3_Done,  T3_9_Done  : BOOL;
    T12_3_Done, T6_9_Done  : BOOL;
    T3_6_Done,  T9_12_Done : BOOL;
    T12_9_Done, T6_3_Done  : BOOL;
    T9_6_Done,  T3_12_Done : BOOL;

    Reset : BOOL;
END_VAR
VAR_OUTPUT
    // Start requests to transfers
    Start_12_6, Start_6_12 : BOOL;
    Start_9_3,  Start_3_9  : BOOL;
    Start_12_3, Start_6_9  : BOOL;
    Start_3_6,  Start_9_12 : BOOL;
    Start_12_9, Start_6_3  : BOOL;
    Start_9_6,  Start_3_12 : BOOL;

    Busy : BOOL;
END_VAR
VAR
    activeRoute : INT := 0; // currently active route ID
END_VAR

// ------------------- MAIN LOGIC -------------------

IF Reset THEN
    Busy := FALSE;
    activeRoute := 0;
END_IF

// --- If not busy, pick a new route ---
IF NOT Busy THEN
    // clear all start outputs
    Start_12_6 := FALSE; Start_6_12 := FALSE;
    Start_9_3  := FALSE; Start_3_9  := FALSE;
    Start_12_3 := FALSE; Start_6_9  := FALSE;
    Start_3_6  := FALSE; Start_9_12 := FALSE;
    Start_12_9 := FALSE; Start_6_3  := FALSE;
    Start_9_6  := FALSE; Start_3_12 := FALSE;

    // check Readers one by one
    IF Reader12_Valid THEN
        CASE Reader12_Value OF
            6:  Start_12_6 := TRUE; activeRoute := 126; Busy := TRUE;
            3:  Start_12_3 := TRUE; activeRoute := 123; Busy := TRUE;
            9:  Start_12_9 := TRUE; activeRoute := 129; Busy := TRUE;
        END_CASE
    ELSIF Reader6_Valid THEN
        CASE Reader6_Value OF
            12: Start_6_12 := TRUE; activeRoute := 612; Busy := TRUE;
            9:  Start_6_9  := TRUE; activeRoute := 69;  Busy := TRUE;
            3:  Start_6_3  := TRUE; activeRoute := 63;  Busy := TRUE;
        END_CASE
    ELSIF Reader3_Valid THEN
        CASE Reader3_Value OF
            9:  Start_3_9  := TRUE; activeRoute := 39;  Busy := TRUE;
            6:  Start_3_6  := TRUE; activeRoute := 36;  Busy := TRUE;
            12: Start_3_12 := TRUE; activeRoute := 312; Busy := TRUE;
        END_CASE
    ELSIF Reader9_Valid THEN
        CASE Reader9_Value OF
            3:  Start_9_3  := TRUE; activeRoute := 93;  Busy := TRUE;
            12: Start_9_12 := TRUE; activeRoute := 912; Busy := TRUE;
            6:  Start_9_6  := TRUE; activeRoute := 96;  Busy := TRUE;
        END_CASE
    END_IF

// --- If busy, wait until the active transfer finishes ---
ELSE
    CASE activeRoute OF
        126: IF T12_6_Done THEN Busy := FALSE; activeRoute := 0; END_IF
        612: IF T6_12_Done THEN Busy := FALSE; activeRoute := 0; END_IF
        93 : IF T9_3_Done  THEN Busy := FALSE; activeRoute := 0; END_IF
        39 : IF T3_9_Done  THEN Busy := FALSE; activeRoute := 0; END_IF
        123: IF T12_3_Done THEN Busy := FALSE; activeRoute := 0; END_IF
        69 : IF T6_9_Done  THEN Busy := FALSE; activeRoute := 0; END_IF
        36 : IF T3_6_Done  THEN Busy := FALSE; activeRoute := 0; END_IF
        912: IF T9_12_Done THEN Busy := FALSE; activeRoute := 0; END_IF
        129: IF T12_9_Done THEN Busy := FALSE; activeRoute := 0; END_IF
        63 : IF T6_3_Done  THEN Busy := FALSE; activeRoute := 0; END_IF
        96 : IF T9_6_Done  THEN Busy := FALSE; activeRoute := 0; END_IF
        312: IF T3_12_Done THEN Busy := FALSE; activeRoute := 0; END_IF
    END_CASE
END_IF

END_FUNCTION_BLOCK

// ---- POUs/FBs/Scheduler/FB_Scheduler_Queue_copy.TcPOU
FUNCTION_BLOCK FB_Scheduler_Queue_copy
VAR_INPUT
    // Reader inputs
    Reader12_Valid : BOOL;
    Reader12_Value : INT;
    Reader3_Valid  : BOOL;
    Reader3_Value  : INT;
    Reader6_Valid  : BOOL;
    Reader6_Value  : INT;
    Reader9_Valid  : BOOL;
    Reader9_Value  : INT;

    // Done flags from transfers
    T12_6_Done, T6_12_Done : BOOL;
    T9_3_Done,  T3_9_Done  : BOOL;
    T12_3_Done, T6_9_Done  : BOOL;
    T3_6_Done,  T9_12_Done : BOOL;
    T12_9_Done, T6_3_Done  : BOOL;
    T9_6_Done,  T3_12_Done : BOOL;

    Reset : BOOL;
END_VAR
VAR_OUTPUT
    // Start signals (1-scan pulses)
    Start_12_6, Start_6_12 : BOOL;
    Start_9_3,  Start_3_9  : BOOL;
    Start_12_3, Start_6_9  : BOOL;
    Start_3_6,  Start_9_12 : BOOL;
    Start_12_9, Start_6_3  : BOOL;
    Start_9_6,  Start_3_12 : BOOL;

    Busy        : BOOL;
    QCount      : INT;     // number of queued requests
    activeRoute : INT;     // currently executing route
END_VAR
VAR
    queue   : ARRAY[1..10] OF INT;   // FIFO buffer (10 deep)
    head    : INT := 1;
    tail    : INT := 1;
	prevR12, prevR3, prevR6, prevR9 : BOOL;
END_VAR

// === Reset ===
IF Reset THEN
    head := 1; tail := 1; QCount := 0;
    Busy := FALSE; activeRoute := 0;
END_IF

// === Enqueue new reader requests ===
IF Reader12_Valid AND NOT prevR12 THEN
    CASE Reader12_Value OF
        6: Enqueue(126);
        3: Enqueue(123);
        9: Enqueue(129);
    END_CASE
END_IF
prevR12 := Reader12_Valid;

IF Reader6_Valid AND NOT prevR6 THEN
    CASE Reader6_Value OF
        12: Enqueue(612);
        9:  Enqueue(69);
        3:  Enqueue(63);
    END_CASE
END_IF
prevR6 := Reader6_Valid;

IF Reader3_Valid AND NOT prevR3 THEN
    CASE Reader3_Value OF
        9:  Enqueue(39);
        6:  Enqueue(36);
        12: Enqueue(312);
    END_CASE
END_IF
prevR3 := Reader3_Valid;

IF Reader9_Valid AND NOT prevR9 THEN
    CASE Reader9_Value OF
        3:  Enqueue(93);
        12: Enqueue(912);
        6:  Enqueue(96);
    END_CASE
END_IF
prevR9 := Reader9_Valid;

// === Dispatch logic (Level Hold) ===
IF NOT Busy AND QCount > 0 THEN
    activeRoute := queue[head];
    head := (head MOD 10) + 1;
    QCount := QCount - 1;
    Busy := TRUE;
END_IF

// Default OFF
Start_12_6 := FALSE; Start_6_12 := FALSE;
Start_9_3  := FALSE; Start_3_9  := FALSE;
Start_12_3 := FALSE; Start_6_9  := FALSE;
Start_3_6  := FALSE; Start_9_12 := FALSE;
Start_12_9 := FALSE; Start_6_3  := FALSE;
Start_9_6  := FALSE; Start_3_12 := FALSE;

// Keep Start HIGH while route is active
CASE activeRoute OF
    126: 
        Start_12_6 := TRUE;
        IF T12_6_Done THEN Busy := FALSE; activeRoute := 0; END_IF
    612: 
        Start_6_12 := TRUE;
        IF T6_12_Done THEN Busy := FALSE; activeRoute := 0; END_IF
    93 : 
        Start_9_3 := TRUE;
        IF T9_3_Done THEN Busy := FALSE; activeRoute := 0; END_IF
    39 : 
        Start_3_9 := TRUE;
        IF T3_9_Done THEN Busy := FALSE; activeRoute := 0; END_IF
    123: 
        Start_12_3 := TRUE;
        IF T12_3_Done THEN Busy := FALSE; activeRoute := 0; END_IF
    69 : 
        Start_6_9 := TRUE;
        IF T6_9_Done THEN Busy := FALSE; activeRoute := 0; END_IF
    36 : 
        Start_3_6 := TRUE;
        IF T3_6_Done THEN Busy := FALSE; activeRoute := 0; END_IF
    912: 
        Start_9_12 := TRUE;
        IF T9_12_Done THEN Busy := FALSE; activeRoute := 0; END_IF
    129: 
        Start_12_9 := TRUE;
        IF T12_9_Done THEN Busy := FALSE; activeRoute := 0; END_IF
    63 : 
        Start_6_3 := TRUE;
        IF T6_3_Done THEN Busy := FALSE; activeRoute := 0; END_IF
    96 : 
        Start_9_6 := TRUE;
        IF T9_6_Done THEN Busy := FALSE; activeRoute := 0; END_IF
    312: 
        Start_3_12 := TRUE;
        IF T3_12_Done THEN Busy := FALSE; activeRoute := 0; END_IF
END_CASE
//// === Dispatch logic ===
//IF NOT Busy AND QCount > 0 THEN
//    activeRoute := queue[head];
//    head := (head MOD 10) + 1;
//    QCount := QCount - 1;
//    Busy := TRUE;

//    // one-shot Start signal
//    CASE activeRoute OF
//        126: Start_12_6 := TRUE;
//        612: Start_6_12 := TRUE;
//        93 : Start_9_3  := TRUE;
//        39 : Start_3_9  := TRUE;
//        123: Start_12_3 := TRUE;
//        69 : Start_6_9  := TRUE;
//        36 : Start_3_6  := TRUE;
//        912: Start_9_12 := TRUE;
//        129: Start_12_9 := TRUE;
//        63 : Start_6_3  := TRUE;
//        96 : Start_9_6  := TRUE;
//        312: Start_3_12 := TRUE;
//    END_CASE
//ELSE
//    Start_12_6 := FALSE; Start_6_12 := FALSE;
//    Start_9_3  := FALSE; Start_3_9  := FALSE;
//    Start_12_3 := FALSE; Start_6_9  := FALSE;
//    Start_3_6  := FALSE; Start_9_12 := FALSE;
//    Start_12_9 := FALSE; Start_6_3  := FALSE;
//    Start_9_6  := FALSE; Start_3_12 := FALSE;
//END_IF


//// === Completion check ===
//CASE activeRoute OF
//    126: IF T12_6_Done THEN Busy := FALSE; activeRoute := 0; END_IF
//    612: IF T6_12_Done THEN Busy := FALSE; activeRoute := 0; END_IF
//    93 : IF T9_3_Done  THEN Busy := FALSE; activeRoute := 0; END_IF
//    39 : IF T3_9_Done  THEN Busy := FALSE; activeRoute := 0; END_IF
//    123: IF T12_3_Done THEN Busy := FALSE; activeRoute := 0; END_IF
//    69 : IF T6_9_Done  THEN Busy := FALSE; activeRoute := 0; END_IF
//    36 : IF T3_6_Done  THEN Busy := FALSE; activeRoute := 0; END_IF
//    912: IF T9_12_Done THEN Busy := FALSE; activeRoute := 0; END_IF
//    129: IF T12_9_Done THEN Busy := FALSE; activeRoute := 0; END_IF
//    63 : IF T6_3_Done  THEN Busy := FALSE; activeRoute := 0; END_IF
//    96 : IF T9_6_Done  THEN Busy := FALSE; activeRoute := 0; END_IF
//    312: IF T3_12_Done THEN Busy := FALSE; activeRoute := 0; END_IF
//END_CASE

METHOD PRIVATE Enqueue : BOOL
VAR_INPUT
    route : INT;
END_VAR

IF QCount < 10 THEN
    queue[tail] := route;
    tail := (tail MOD 10) + 1;
    QCount := QCount + 1;
    Enqueue := TRUE;
ELSE
    Enqueue := FALSE; // queue full
END_IF
END_METHOD

END_FUNCTION_BLOCK
